// TwinCAT 3 PLC project plc_lamp_lv17_vac
// ProgramVersion: 3.1.4022.7
// CompilerDefines: VISU_USEPROPERTYINFO
// libraries:
//   LCLS General, * (SLAC)
//   PMPS, * (SLAC - LCLS)
//   Tc2_SerialCom, * (Beckhoff Automation GmbH)
//   Tc2_Standard, * (Beckhoff Automation GmbH)
//   Tc2_System, * (Beckhoff Automation GmbH)
//   Tc3_Module, * (Beckhoff Automation GmbH)
//   LCLS Vacuum,1.4.0,SLAC - LCLS
//   LCLSVacuumSerialDriverLib,1.2.2,SLAC - LCLS
// project tree:
//   / ComTask.TcTTO (not stored), GlobalTextList.TcGTLO (not stored), PlcTask.TcTTO (not stored)
//   GVLs/ GVL_COM.TcGVL, GVL_Devices.TcGVL, GVL_PLC_Interfaces.TcGVL (not stored), GVL_Variables.TcGVL (not stored)
//   POUs/ DIAGNOSTICS.TcPOU (not stored), F_Turbo_NC_NO_Valve_Logic.TcPOU (not stored), MAIN.TcPOU, PRG_COM.TcPOU
// real-time tasks:
//   TASK PlcTask: cycle T#10ms, priority 20, ADS port 350
//   TASK ComTask: cycle T#10ms, priority 15, ADS port 351
// I/O:
//   DEVICE Device 1 (EtherCAT), AmsNetId 172.21.132.34.2.1
//     LAMP_PLC_E0_EK1200 [EK1200-5000 EtherCAT Power supply (2A E-Bus)]
//       LAMP_PLC_E1_EL2202
//       LAMP_PLC_E2_EL6070
//       LAMP_PLC_E3_EL6692 [EL6692 EtherCAT Bridge terminal (Primary)]
//       LAMP_PLC_E4_EL9410
//       LAMP_PLC_E5_EL1004
//       LAMP_PLC_E6_EL2794
//       LAMP_PLC_E7_EL1004
//       LAMP_PLC_E8_EL2794
//       LAMP_PLC_E9_EL3318 [EL3318 8Ch. Ana Input Thermocouple (TC)]
//       LAMP_PLC_E10_EL6002
//       LAMP_PLC_E11_EL6002
//       LAMP_PLC_E12_EK1122 [EK1122 2 port EtherCAT junction]
//         LAMP_PNL_EP00_EP9128-0021 [EP9128-0021 8x EtherCAT junction]
//           LAMP_PNL1_EP01_EP2338-0002
//           LAMP_PNL1_EP02_EP2624-0002
//           LAMP_PNL1_EP03_EP6002-0002
//           LAMP_PNL1_EP04_EP2338-0002
//           LAMP_PNL1_EP05_EP2624-0002
//           LAMP_PNL1_EP06_EP6002-0002
//           LAMP_PNL1_EP07_EP2338-0002
//           LAMP_PNL1_EP08_EP2624-0002
//           LAMP_PNL1_EP09_EP6002-0002
//           LAMP_PNL1_EP10_EP2338-0002
//           LAMP_PNL1_EP11_EP2624-0002
//           LAMP_PNL1_EP12_EP6002-0002
//           LAMP_PNL2_EP13_EP2338-0002
//           LAMP_PNL2_EP14_EP2624-0002
//           LAMP_PNL2_EP15_EP6002-0002
//           LAMP_PNL2_EP16_EP2338-0002
//           LAMP_PNL2_EP17_EP2624-0002
//           LAMP_PN2_EP18_EP6002-0002
//           LAMP_PNL2_EP19_EP3174-0002
//           LAMP_PNL2_EP20_EP3174-0002
//           LAMP_PNL2_EP21_EP3174-0002
//           LAMP_PNL2_EP22_EP2624-0002
//           LAMP_PNL2_EP23_EP3174-0002
//           LAMP_PNL2_EP24_EP2624-0002
//           LAMP_PNL2_EP25_EP2338-0002
//           LAMP_PNL2_EP26_EP2338-0002
//           Term 88 (EP9128-1021) [EP9128-1021 8x EtherCAT junction - Dev A]
//             LAMP_CLSTR1_PNL1_EP01_EP2338-0002
//             LAMP_CLSTR1_PNL1_EP_02_EP2624-0002
//             LAMP_CLSTR1_PNL1_EP03_EP6002-0002
//             LAMP_CLSTR1_PNL3_EP01_EP2338-0002
//             LAMP_CLSTR1_PNL3_EP02_EP2624-0002
//             LAMP_CLSTR1_PNL3_EP03_EP6002-0002
//           Term 89 (EP9128-2021) [EP9128-2021 8x EtherCAT junction - Dev B]
//             LAMP_CLSTR1_PNL2_EP01_EP2338-0002
//             LAMP_CLSTR1_PNL2_EP02_EP2624-0002
//             LAMP_CLSTR1_PNL2_EP03_EP6002-0002
//             LAMP_CLSTR1_DCT_EP9224-0023
//         LAMP_PNL1_PWR_FOUT_Box (EP9224-0023) [EP9224-0023 4Ch/4Ch enhanced Power Distribution for EtherCAT Box Modules]
// variable links:
//   plc_lamp_lv17_vac/plc_lamp_lv17_vac Instance <-> Device 1 (EtherCAT)/LAMP_PLC_E0_EK1200/LAMP_PLC_E12_EK1122/LAMP_PNL_EP00_EP9128-0021/LAMP_PNL1_EP01_EP2338-0002
//     PlcTask Inputs/GVL_Devices.LAMP_C2_PTM_01.i_xAtSpd <-> Channel 1/Input
//     PlcTask Inputs/GVL_Devices.LAMP_C2_PTM_02.i_xAtSpd <-> Channel 5/Input
//     PlcTask Inputs/GVL_Devices.LAMP_C2_PTM_01.i_xFaultNC <-> Channel 2/Input
//     PlcTask Inputs/GVL_Devices.LAMP_C2_PTM_02.i_xFaultNC <-> Channel 6/Input
//     PlcTask Inputs/GVL_Devices.LAMP_C2_PTM_01.i_xRemote <-> Channel 3/Input
//     PlcTask Inputs/GVL_Devices.LAMP_C2_PTM_02.i_xRemote <-> Channel 7/Input
//   plc_lamp_lv17_vac/plc_lamp_lv17_vac Instance <-> Device 1 (EtherCAT)/LAMP_PLC_E0_EK1200/LAMP_PLC_E12_EK1122/LAMP_PNL_EP00_EP9128-0021/LAMP_PNL1_EP02_EP2624-0002
//     PlcTask Outputs/GVL_Devices.LAMP_C2_PTM_01.q_RunDO <-> Channel 1/Output
//     PlcTask Outputs/GVL_Devices.LAMP_C2_PTM_02.q_RunDO <-> Channel 3/Output
//     PlcTask Outputs/GVL_Devices.LAMP_C2_PTM_01.q_xReset <-> Channel 2/Output
//     PlcTask Outputs/GVL_Devices.LAMP_C2_PTM_02.q_xReset <-> Channel 4/Output
//   plc_lamp_lv17_vac/plc_lamp_lv17_vac Instance <-> Device 1 (EtherCAT)/LAMP_PLC_E0_EK1200/LAMP_PLC_E12_EK1122/LAMP_PNL_EP00_EP9128-0021/LAMP_PNL1_EP03_EP6002-0002
//     ComTask Inputs/GVL_COM.stComIn_LAMP_C2_PTM_01/D[0] <-> COM TxPDO-Map Inputs Channel 1/Data In 0
//     ComTask Inputs/GVL_COM.stComIn_LAMP_C2_PTM_01/D[10] <-> COM TxPDO-Map Inputs Channel 1/Data In 10
//     ComTask Inputs/GVL_COM.stComIn_LAMP_C2_PTM_01/D[11] <-> COM TxPDO-Map Inputs Channel 1/Data In 11
//     ComTask Inputs/GVL_COM.stComIn_LAMP_C2_PTM_01/D[12] <-> COM TxPDO-Map Inputs Channel 1/Data In 12
//     ComTask Inputs/GVL_COM.stComIn_LAMP_C2_PTM_01/D[13] <-> COM TxPDO-Map Inputs Channel 1/Data In 13
//     ComTask Inputs/GVL_COM.stComIn_LAMP_C2_PTM_01/D[14] <-> COM TxPDO-Map Inputs Channel 1/Data In 14
//     ComTask Inputs/GVL_COM.stComIn_LAMP_C2_PTM_01/D[15] <-> COM TxPDO-Map Inputs Channel 1/Data In 15
//     ComTask Inputs/GVL_COM.stComIn_LAMP_C2_PTM_01/D[16] <-> COM TxPDO-Map Inputs Channel 1/Data In 16
//     ComTask Inputs/GVL_COM.stComIn_LAMP_C2_PTM_01/D[17] <-> COM TxPDO-Map Inputs Channel 1/Data In 17
//     ComTask Inputs/GVL_COM.stComIn_LAMP_C2_PTM_01/D[18] <-> COM TxPDO-Map Inputs Channel 1/Data In 18
//     ComTask Inputs/GVL_COM.stComIn_LAMP_C2_PTM_01/D[19] <-> COM TxPDO-Map Inputs Channel 1/Data In 19
//     ComTask Inputs/GVL_COM.stComIn_LAMP_C2_PTM_01/D[1] <-> COM TxPDO-Map Inputs Channel 1/Data In 1
//     ComTask Inputs/GVL_COM.stComIn_LAMP_C2_PTM_01/D[20] <-> COM TxPDO-Map Inputs Channel 1/Data In 20
//     ComTask Inputs/GVL_COM.stComIn_LAMP_C2_PTM_01/D[21] <-> COM TxPDO-Map Inputs Channel 1/Data In 21
//     ComTask Inputs/GVL_COM.stComIn_LAMP_C2_PTM_01/D[2] <-> COM TxPDO-Map Inputs Channel 1/Data In 2
//     ComTask Inputs/GVL_COM.stComIn_LAMP_C2_PTM_01/D[3] <-> COM TxPDO-Map Inputs Channel 1/Data In 3
//     ComTask Inputs/GVL_COM.stComIn_LAMP_C2_PTM_01/D[4] <-> COM TxPDO-Map Inputs Channel 1/Data In 4
//     ComTask Inputs/GVL_COM.stComIn_LAMP_C2_PTM_01/D[5] <-> COM TxPDO-Map Inputs Channel 1/Data In 5
//     ComTask Inputs/GVL_COM.stComIn_LAMP_C2_PTM_01/D[6] <-> COM TxPDO-Map Inputs Channel 1/Data In 6
//     ComTask Inputs/GVL_COM.stComIn_LAMP_C2_PTM_01/D[7] <-> COM TxPDO-Map Inputs Channel 1/Data In 7
//     ComTask Inputs/GVL_COM.stComIn_LAMP_C2_PTM_01/D[8] <-> COM TxPDO-Map Inputs Channel 1/Data In 8
//     ComTask Inputs/GVL_COM.stComIn_LAMP_C2_PTM_01/D[9] <-> COM TxPDO-Map Inputs Channel 1/Data In 9
//     ComTask Inputs/GVL_COM.stComIn_LAMP_C2_PTM_02/D[0] <-> COM TxPDO-Map Inputs Channel 2/Data In 0
//     ComTask Inputs/GVL_COM.stComIn_LAMP_C2_PTM_02/D[10] <-> COM TxPDO-Map Inputs Channel 2/Data In 10
//     ComTask Inputs/GVL_COM.stComIn_LAMP_C2_PTM_02/D[11] <-> COM TxPDO-Map Inputs Channel 2/Data In 11
//     ComTask Inputs/GVL_COM.stComIn_LAMP_C2_PTM_02/D[12] <-> COM TxPDO-Map Inputs Channel 2/Data In 12
//     ComTask Inputs/GVL_COM.stComIn_LAMP_C2_PTM_02/D[13] <-> COM TxPDO-Map Inputs Channel 2/Data In 13
//     ComTask Inputs/GVL_COM.stComIn_LAMP_C2_PTM_02/D[14] <-> COM TxPDO-Map Inputs Channel 2/Data In 14
//     ComTask Inputs/GVL_COM.stComIn_LAMP_C2_PTM_02/D[15] <-> COM TxPDO-Map Inputs Channel 2/Data In 15
//     ComTask Inputs/GVL_COM.stComIn_LAMP_C2_PTM_02/D[16] <-> COM TxPDO-Map Inputs Channel 2/Data In 16
//     ComTask Inputs/GVL_COM.stComIn_LAMP_C2_PTM_02/D[17] <-> COM TxPDO-Map Inputs Channel 2/Data In 17
//     ComTask Inputs/GVL_COM.stComIn_LAMP_C2_PTM_02/D[18] <-> COM TxPDO-Map Inputs Channel 2/Data In 18
//     ComTask Inputs/GVL_COM.stComIn_LAMP_C2_PTM_02/D[19] <-> COM TxPDO-Map Inputs Channel 2/Data In 19
//     ComTask Inputs/GVL_COM.stComIn_LAMP_C2_PTM_02/D[1] <-> COM TxPDO-Map Inputs Channel 2/Data In 1
//     ComTask Inputs/GVL_COM.stComIn_LAMP_C2_PTM_02/D[20] <-> COM TxPDO-Map Inputs Channel 2/Data In 20
//     ComTask Inputs/GVL_COM.stComIn_LAMP_C2_PTM_02/D[21] <-> COM TxPDO-Map Inputs Channel 2/Data In 21
//     ComTask Inputs/GVL_COM.stComIn_LAMP_C2_PTM_02/D[2] <-> COM TxPDO-Map Inputs Channel 2/Data In 2
//     ComTask Inputs/GVL_COM.stComIn_LAMP_C2_PTM_02/D[3] <-> COM TxPDO-Map Inputs Channel 2/Data In 3
//     ComTask Inputs/GVL_COM.stComIn_LAMP_C2_PTM_02/D[4] <-> COM TxPDO-Map Inputs Channel 2/Data In 4
//     ComTask Inputs/GVL_COM.stComIn_LAMP_C2_PTM_02/D[5] <-> COM TxPDO-Map Inputs Channel 2/Data In 5
//     ComTask Inputs/GVL_COM.stComIn_LAMP_C2_PTM_02/D[6] <-> COM TxPDO-Map Inputs Channel 2/Data In 6
//     ComTask Inputs/GVL_COM.stComIn_LAMP_C2_PTM_02/D[7] <-> COM TxPDO-Map Inputs Channel 2/Data In 7
//     ComTask Inputs/GVL_COM.stComIn_LAMP_C2_PTM_02/D[8] <-> COM TxPDO-Map Inputs Channel 2/Data In 8
//     ComTask Inputs/GVL_COM.stComIn_LAMP_C2_PTM_02/D[9] <-> COM TxPDO-Map Inputs Channel 2/Data In 9
//     ComTask Inputs/GVL_COM.stComIn_LAMP_C2_PTM_01/Status <-> COM TxPDO-Map Inputs Channel 1/Status
//     ComTask Inputs/GVL_COM.stComIn_LAMP_C2_PTM_02/Status <-> COM TxPDO-Map Inputs Channel 2/Status
//     ComTask Outputs/GVL_COM.stComOut_LAMP_C2_PTM_01/Ctrl <-> COM RxPDO-Map Outputs Channel 1/Ctrl
//     ComTask Outputs/GVL_COM.stComOut_LAMP_C2_PTM_02/Ctrl <-> COM RxPDO-Map Outputs Channel 2/Ctrl
//     ComTask Outputs/GVL_COM.stComOut_LAMP_C2_PTM_01/D[0] <-> COM RxPDO-Map Outputs Channel 1/Data Out 0
//     ComTask Outputs/GVL_COM.stComOut_LAMP_C2_PTM_01/D[10] <-> COM RxPDO-Map Outputs Channel 1/Data Out 10
//     ComTask Outputs/GVL_COM.stComOut_LAMP_C2_PTM_01/D[11] <-> COM RxPDO-Map Outputs Channel 1/Data Out 11
//     ComTask Outputs/GVL_COM.stComOut_LAMP_C2_PTM_01/D[12] <-> COM RxPDO-Map Outputs Channel 1/Data Out 12
//     ComTask Outputs/GVL_COM.stComOut_LAMP_C2_PTM_01/D[13] <-> COM RxPDO-Map Outputs Channel 1/Data Out 13
//     ComTask Outputs/GVL_COM.stComOut_LAMP_C2_PTM_01/D[14] <-> COM RxPDO-Map Outputs Channel 1/Data Out 14
//     ComTask Outputs/GVL_COM.stComOut_LAMP_C2_PTM_01/D[15] <-> COM RxPDO-Map Outputs Channel 1/Data Out 15
//     ComTask Outputs/GVL_COM.stComOut_LAMP_C2_PTM_01/D[16] <-> COM RxPDO-Map Outputs Channel 1/Data Out 16
//     ComTask Outputs/GVL_COM.stComOut_LAMP_C2_PTM_01/D[17] <-> COM RxPDO-Map Outputs Channel 1/Data Out 17
//     ComTask Outputs/GVL_COM.stComOut_LAMP_C2_PTM_01/D[18] <-> COM RxPDO-Map Outputs Channel 1/Data Out 18
//     ComTask Outputs/GVL_COM.stComOut_LAMP_C2_PTM_01/D[19] <-> COM RxPDO-Map Outputs Channel 1/Data Out 19
//     ComTask Outputs/GVL_COM.stComOut_LAMP_C2_PTM_01/D[1] <-> COM RxPDO-Map Outputs Channel 1/Data Out 1
//     ComTask Outputs/GVL_COM.stComOut_LAMP_C2_PTM_01/D[20] <-> COM RxPDO-Map Outputs Channel 1/Data Out 20
//     ComTask Outputs/GVL_COM.stComOut_LAMP_C2_PTM_01/D[21] <-> COM RxPDO-Map Outputs Channel 1/Data Out 21
//     ComTask Outputs/GVL_COM.stComOut_LAMP_C2_PTM_01/D[2] <-> COM RxPDO-Map Outputs Channel 1/Data Out 2
//     ComTask Outputs/GVL_COM.stComOut_LAMP_C2_PTM_01/D[3] <-> COM RxPDO-Map Outputs Channel 1/Data Out 3
//     ComTask Outputs/GVL_COM.stComOut_LAMP_C2_PTM_01/D[4] <-> COM RxPDO-Map Outputs Channel 1/Data Out 4
//     ComTask Outputs/GVL_COM.stComOut_LAMP_C2_PTM_01/D[5] <-> COM RxPDO-Map Outputs Channel 1/Data Out 5
//     ComTask Outputs/GVL_COM.stComOut_LAMP_C2_PTM_01/D[6] <-> COM RxPDO-Map Outputs Channel 1/Data Out 6
//     ComTask Outputs/GVL_COM.stComOut_LAMP_C2_PTM_01/D[7] <-> COM RxPDO-Map Outputs Channel 1/Data Out 7
//     ComTask Outputs/GVL_COM.stComOut_LAMP_C2_PTM_01/D[8] <-> COM RxPDO-Map Outputs Channel 1/Data Out 8
//     ComTask Outputs/GVL_COM.stComOut_LAMP_C2_PTM_01/D[9] <-> COM RxPDO-Map Outputs Channel 1/Data Out 9
//     ComTask Outputs/GVL_COM.stComOut_LAMP_C2_PTM_02/D[0] <-> COM RxPDO-Map Outputs Channel 2/Data Out 0
//     ComTask Outputs/GVL_COM.stComOut_LAMP_C2_PTM_02/D[10] <-> COM RxPDO-Map Outputs Channel 2/Data Out 10
//     ComTask Outputs/GVL_COM.stComOut_LAMP_C2_PTM_02/D[11] <-> COM RxPDO-Map Outputs Channel 2/Data Out 11
//     ComTask Outputs/GVL_COM.stComOut_LAMP_C2_PTM_02/D[12] <-> COM RxPDO-Map Outputs Channel 2/Data Out 12
//     ComTask Outputs/GVL_COM.stComOut_LAMP_C2_PTM_02/D[13] <-> COM RxPDO-Map Outputs Channel 2/Data Out 13
//     ComTask Outputs/GVL_COM.stComOut_LAMP_C2_PTM_02/D[14] <-> COM RxPDO-Map Outputs Channel 2/Data Out 14
//     ComTask Outputs/GVL_COM.stComOut_LAMP_C2_PTM_02/D[15] <-> COM RxPDO-Map Outputs Channel 2/Data Out 15
//     ComTask Outputs/GVL_COM.stComOut_LAMP_C2_PTM_02/D[16] <-> COM RxPDO-Map Outputs Channel 2/Data Out 16
//     ComTask Outputs/GVL_COM.stComOut_LAMP_C2_PTM_02/D[17] <-> COM RxPDO-Map Outputs Channel 2/Data Out 17
//     ComTask Outputs/GVL_COM.stComOut_LAMP_C2_PTM_02/D[18] <-> COM RxPDO-Map Outputs Channel 2/Data Out 18
//     ComTask Outputs/GVL_COM.stComOut_LAMP_C2_PTM_02/D[19] <-> COM RxPDO-Map Outputs Channel 2/Data Out 19
//     ComTask Outputs/GVL_COM.stComOut_LAMP_C2_PTM_02/D[1] <-> COM RxPDO-Map Outputs Channel 2/Data Out 1
//     ComTask Outputs/GVL_COM.stComOut_LAMP_C2_PTM_02/D[20] <-> COM RxPDO-Map Outputs Channel 2/Data Out 20
//     ComTask Outputs/GVL_COM.stComOut_LAMP_C2_PTM_02/D[21] <-> COM RxPDO-Map Outputs Channel 2/Data Out 21
//     ComTask Outputs/GVL_COM.stComOut_LAMP_C2_PTM_02/D[2] <-> COM RxPDO-Map Outputs Channel 2/Data Out 2
//     ComTask Outputs/GVL_COM.stComOut_LAMP_C2_PTM_02/D[3] <-> COM RxPDO-Map Outputs Channel 2/Data Out 3
//     ComTask Outputs/GVL_COM.stComOut_LAMP_C2_PTM_02/D[4] <-> COM RxPDO-Map Outputs Channel 2/Data Out 4
//     ComTask Outputs/GVL_COM.stComOut_LAMP_C2_PTM_02/D[5] <-> COM RxPDO-Map Outputs Channel 2/Data Out 5
//     ComTask Outputs/GVL_COM.stComOut_LAMP_C2_PTM_02/D[6] <-> COM RxPDO-Map Outputs Channel 2/Data Out 6
//     ComTask Outputs/GVL_COM.stComOut_LAMP_C2_PTM_02/D[7] <-> COM RxPDO-Map Outputs Channel 2/Data Out 7
//     ComTask Outputs/GVL_COM.stComOut_LAMP_C2_PTM_02/D[8] <-> COM RxPDO-Map Outputs Channel 2/Data Out 8
//     ComTask Outputs/GVL_COM.stComOut_LAMP_C2_PTM_02/D[9] <-> COM RxPDO-Map Outputs Channel 2/Data Out 9
//   plc_lamp_lv17_vac/plc_lamp_lv17_vac Instance <-> Device 1 (EtherCAT)/LAMP_PLC_E0_EK1200/LAMP_PLC_E12_EK1122/LAMP_PNL_EP00_EP9128-0021/LAMP_PNL1_EP04_EP2338-0002
//     PlcTask Inputs/GVL_Devices.LAMP_C2_PTM_03.i_xAtSpd <-> Channel 1/Input
//     PlcTask Inputs/GVL_Devices.LAMP_C2_PTM_04.i_xAtSpd <-> Channel 5/Input
//     PlcTask Inputs/GVL_Devices.LAMP_C2_PTM_03.i_xFaultNC <-> Channel 2/Input
//     PlcTask Inputs/GVL_Devices.LAMP_C2_PTM_04.i_xFaultNC <-> Channel 6/Input
//     PlcTask Inputs/GVL_Devices.LAMP_C2_PTM_03.i_xRemote <-> Channel 3/Input
//     PlcTask Inputs/GVL_Devices.LAMP_C2_PTM_04.i_xRemote <-> Channel 7/Input
//   plc_lamp_lv17_vac/plc_lamp_lv17_vac Instance <-> Device 1 (EtherCAT)/LAMP_PLC_E0_EK1200/LAMP_PLC_E12_EK1122/LAMP_PNL_EP00_EP9128-0021/LAMP_PNL1_EP05_EP2624-0002
//     PlcTask Outputs/GVL_Devices.LAMP_C2_PTM_03.q_RunDO <-> Channel 1/Output
//     PlcTask Outputs/GVL_Devices.LAMP_C2_PTM_04.q_RunDO <-> Channel 3/Output
//     PlcTask Outputs/GVL_Devices.LAMP_C2_PTM_03.q_xReset <-> Channel 2/Output
//     PlcTask Outputs/GVL_Devices.LAMP_C2_PTM_04.q_xReset <-> Channel 4/Output
//   plc_lamp_lv17_vac/plc_lamp_lv17_vac Instance <-> Device 1 (EtherCAT)/LAMP_PLC_E0_EK1200/LAMP_PLC_E12_EK1122/LAMP_PNL_EP00_EP9128-0021/LAMP_PNL1_EP06_EP6002-0002
//     ComTask Inputs/GVL_COM.stComIn_LAMP_C2_PTM_03/D[0] <-> COM TxPDO-Map Inputs Channel 1/Data In 0
//     ComTask Inputs/GVL_COM.stComIn_LAMP_C2_PTM_03/D[10] <-> COM TxPDO-Map Inputs Channel 1/Data In 10
//     ComTask Inputs/GVL_COM.stComIn_LAMP_C2_PTM_03/D[11] <-> COM TxPDO-Map Inputs Channel 1/Data In 11
//     ComTask Inputs/GVL_COM.stComIn_LAMP_C2_PTM_03/D[12] <-> COM TxPDO-Map Inputs Channel 1/Data In 12
//     ComTask Inputs/GVL_COM.stComIn_LAMP_C2_PTM_03/D[13] <-> COM TxPDO-Map Inputs Channel 1/Data In 13
//     ComTask Inputs/GVL_COM.stComIn_LAMP_C2_PTM_03/D[14] <-> COM TxPDO-Map Inputs Channel 1/Data In 14
//     ComTask Inputs/GVL_COM.stComIn_LAMP_C2_PTM_03/D[15] <-> COM TxPDO-Map Inputs Channel 1/Data In 15
//     ComTask Inputs/GVL_COM.stComIn_LAMP_C2_PTM_03/D[16] <-> COM TxPDO-Map Inputs Channel 1/Data In 16
//     ComTask Inputs/GVL_COM.stComIn_LAMP_C2_PTM_03/D[17] <-> COM TxPDO-Map Inputs Channel 1/Data In 17
//     ComTask Inputs/GVL_COM.stComIn_LAMP_C2_PTM_03/D[18] <-> COM TxPDO-Map Inputs Channel 1/Data In 18
//     ComTask Inputs/GVL_COM.stComIn_LAMP_C2_PTM_03/D[19] <-> COM TxPDO-Map Inputs Channel 1/Data In 19
//     ComTask Inputs/GVL_COM.stComIn_LAMP_C2_PTM_03/D[1] <-> COM TxPDO-Map Inputs Channel 1/Data In 1
//     ComTask Inputs/GVL_COM.stComIn_LAMP_C2_PTM_03/D[20] <-> COM TxPDO-Map Inputs Channel 1/Data In 20
//     ComTask Inputs/GVL_COM.stComIn_LAMP_C2_PTM_03/D[21] <-> COM TxPDO-Map Inputs Channel 1/Data In 21
//     ComTask Inputs/GVL_COM.stComIn_LAMP_C2_PTM_03/D[2] <-> COM TxPDO-Map Inputs Channel 1/Data In 2
//     ComTask Inputs/GVL_COM.stComIn_LAMP_C2_PTM_03/D[3] <-> COM TxPDO-Map Inputs Channel 1/Data In 3
//     ComTask Inputs/GVL_COM.stComIn_LAMP_C2_PTM_03/D[4] <-> COM TxPDO-Map Inputs Channel 1/Data In 4
//     ComTask Inputs/GVL_COM.stComIn_LAMP_C2_PTM_03/D[5] <-> COM TxPDO-Map Inputs Channel 1/Data In 5
//     ComTask Inputs/GVL_COM.stComIn_LAMP_C2_PTM_03/D[6] <-> COM TxPDO-Map Inputs Channel 1/Data In 6
//     ComTask Inputs/GVL_COM.stComIn_LAMP_C2_PTM_03/D[7] <-> COM TxPDO-Map Inputs Channel 1/Data In 7
//     ComTask Inputs/GVL_COM.stComIn_LAMP_C2_PTM_03/D[8] <-> COM TxPDO-Map Inputs Channel 1/Data In 8
//     ComTask Inputs/GVL_COM.stComIn_LAMP_C2_PTM_03/D[9] <-> COM TxPDO-Map Inputs Channel 1/Data In 9
//     ComTask Inputs/GVL_COM.stComIn_LAMP_C2_PTM_04/D[0] <-> COM TxPDO-Map Inputs Channel 2/Data In 0
//     ComTask Inputs/GVL_COM.stComIn_LAMP_C2_PTM_04/D[10] <-> COM TxPDO-Map Inputs Channel 2/Data In 10
//     ComTask Inputs/GVL_COM.stComIn_LAMP_C2_PTM_04/D[11] <-> COM TxPDO-Map Inputs Channel 2/Data In 11
//     ComTask Inputs/GVL_COM.stComIn_LAMP_C2_PTM_04/D[12] <-> COM TxPDO-Map Inputs Channel 2/Data In 12
//     ComTask Inputs/GVL_COM.stComIn_LAMP_C2_PTM_04/D[13] <-> COM TxPDO-Map Inputs Channel 2/Data In 13
//     ComTask Inputs/GVL_COM.stComIn_LAMP_C2_PTM_04/D[14] <-> COM TxPDO-Map Inputs Channel 2/Data In 14
//     ComTask Inputs/GVL_COM.stComIn_LAMP_C2_PTM_04/D[15] <-> COM TxPDO-Map Inputs Channel 2/Data In 15
//     ComTask Inputs/GVL_COM.stComIn_LAMP_C2_PTM_04/D[16] <-> COM TxPDO-Map Inputs Channel 2/Data In 16
//     ComTask Inputs/GVL_COM.stComIn_LAMP_C2_PTM_04/D[17] <-> COM TxPDO-Map Inputs Channel 2/Data In 17
//     ComTask Inputs/GVL_COM.stComIn_LAMP_C2_PTM_04/D[18] <-> COM TxPDO-Map Inputs Channel 2/Data In 18
//     ComTask Inputs/GVL_COM.stComIn_LAMP_C2_PTM_04/D[19] <-> COM TxPDO-Map Inputs Channel 2/Data In 19
//     ComTask Inputs/GVL_COM.stComIn_LAMP_C2_PTM_04/D[1] <-> COM TxPDO-Map Inputs Channel 2/Data In 1
//     ComTask Inputs/GVL_COM.stComIn_LAMP_C2_PTM_04/D[20] <-> COM TxPDO-Map Inputs Channel 2/Data In 20
//     ComTask Inputs/GVL_COM.stComIn_LAMP_C2_PTM_04/D[21] <-> COM TxPDO-Map Inputs Channel 2/Data In 21
//     ComTask Inputs/GVL_COM.stComIn_LAMP_C2_PTM_04/D[2] <-> COM TxPDO-Map Inputs Channel 2/Data In 2
//     ComTask Inputs/GVL_COM.stComIn_LAMP_C2_PTM_04/D[3] <-> COM TxPDO-Map Inputs Channel 2/Data In 3
//     ComTask Inputs/GVL_COM.stComIn_LAMP_C2_PTM_04/D[4] <-> COM TxPDO-Map Inputs Channel 2/Data In 4
//     ComTask Inputs/GVL_COM.stComIn_LAMP_C2_PTM_04/D[5] <-> COM TxPDO-Map Inputs Channel 2/Data In 5
//     ComTask Inputs/GVL_COM.stComIn_LAMP_C2_PTM_04/D[6] <-> COM TxPDO-Map Inputs Channel 2/Data In 6
//     ComTask Inputs/GVL_COM.stComIn_LAMP_C2_PTM_04/D[7] <-> COM TxPDO-Map Inputs Channel 2/Data In 7
//     ComTask Inputs/GVL_COM.stComIn_LAMP_C2_PTM_04/D[8] <-> COM TxPDO-Map Inputs Channel 2/Data In 8
//     ComTask Inputs/GVL_COM.stComIn_LAMP_C2_PTM_04/D[9] <-> COM TxPDO-Map Inputs Channel 2/Data In 9
//     ComTask Inputs/GVL_COM.stComIn_LAMP_C2_PTM_03/Status <-> COM TxPDO-Map Inputs Channel 1/Status
//     ComTask Inputs/GVL_COM.stComIn_LAMP_C2_PTM_04/Status <-> COM TxPDO-Map Inputs Channel 2/Status
//     ComTask Outputs/GVL_COM.stComOut_LAMP_C2_PTM_03/Ctrl <-> COM RxPDO-Map Outputs Channel 1/Ctrl
//     ComTask Outputs/GVL_COM.stComOut_LAMP_C2_PTM_04/Ctrl <-> COM RxPDO-Map Outputs Channel 2/Ctrl
//     ComTask Outputs/GVL_COM.stComOut_LAMP_C2_PTM_03/D[0] <-> COM RxPDO-Map Outputs Channel 1/Data Out 0
//     ComTask Outputs/GVL_COM.stComOut_LAMP_C2_PTM_03/D[10] <-> COM RxPDO-Map Outputs Channel 1/Data Out 10
//     ComTask Outputs/GVL_COM.stComOut_LAMP_C2_PTM_03/D[11] <-> COM RxPDO-Map Outputs Channel 1/Data Out 11
//     ComTask Outputs/GVL_COM.stComOut_LAMP_C2_PTM_03/D[12] <-> COM RxPDO-Map Outputs Channel 1/Data Out 12
//     ComTask Outputs/GVL_COM.stComOut_LAMP_C2_PTM_03/D[13] <-> COM RxPDO-Map Outputs Channel 1/Data Out 13
//     ComTask Outputs/GVL_COM.stComOut_LAMP_C2_PTM_03/D[14] <-> COM RxPDO-Map Outputs Channel 1/Data Out 14
//     ComTask Outputs/GVL_COM.stComOut_LAMP_C2_PTM_03/D[15] <-> COM RxPDO-Map Outputs Channel 1/Data Out 15
//     ComTask Outputs/GVL_COM.stComOut_LAMP_C2_PTM_03/D[16] <-> COM RxPDO-Map Outputs Channel 1/Data Out 16
//     ComTask Outputs/GVL_COM.stComOut_LAMP_C2_PTM_03/D[17] <-> COM RxPDO-Map Outputs Channel 1/Data Out 17
//     ComTask Outputs/GVL_COM.stComOut_LAMP_C2_PTM_03/D[18] <-> COM RxPDO-Map Outputs Channel 1/Data Out 18
//     ComTask Outputs/GVL_COM.stComOut_LAMP_C2_PTM_03/D[19] <-> COM RxPDO-Map Outputs Channel 1/Data Out 19
//     ComTask Outputs/GVL_COM.stComOut_LAMP_C2_PTM_03/D[1] <-> COM RxPDO-Map Outputs Channel 1/Data Out 1
//     ComTask Outputs/GVL_COM.stComOut_LAMP_C2_PTM_03/D[20] <-> COM RxPDO-Map Outputs Channel 1/Data Out 20
//     ComTask Outputs/GVL_COM.stComOut_LAMP_C2_PTM_03/D[21] <-> COM RxPDO-Map Outputs Channel 1/Data Out 21
//     ComTask Outputs/GVL_COM.stComOut_LAMP_C2_PTM_03/D[2] <-> COM RxPDO-Map Outputs Channel 1/Data Out 2
//     ComTask Outputs/GVL_COM.stComOut_LAMP_C2_PTM_03/D[3] <-> COM RxPDO-Map Outputs Channel 1/Data Out 3
//     ComTask Outputs/GVL_COM.stComOut_LAMP_C2_PTM_03/D[4] <-> COM RxPDO-Map Outputs Channel 1/Data Out 4
//     ComTask Outputs/GVL_COM.stComOut_LAMP_C2_PTM_03/D[5] <-> COM RxPDO-Map Outputs Channel 1/Data Out 5
//     ComTask Outputs/GVL_COM.stComOut_LAMP_C2_PTM_03/D[6] <-> COM RxPDO-Map Outputs Channel 1/Data Out 6
//     ComTask Outputs/GVL_COM.stComOut_LAMP_C2_PTM_03/D[7] <-> COM RxPDO-Map Outputs Channel 1/Data Out 7
//     ComTask Outputs/GVL_COM.stComOut_LAMP_C2_PTM_03/D[8] <-> COM RxPDO-Map Outputs Channel 1/Data Out 8
//     ComTask Outputs/GVL_COM.stComOut_LAMP_C2_PTM_03/D[9] <-> COM RxPDO-Map Outputs Channel 1/Data Out 9
//     ComTask Outputs/GVL_COM.stComOut_LAMP_C2_PTM_04/D[0] <-> COM RxPDO-Map Outputs Channel 2/Data Out 0
//     ComTask Outputs/GVL_COM.stComOut_LAMP_C2_PTM_04/D[10] <-> COM RxPDO-Map Outputs Channel 2/Data Out 10
//     ComTask Outputs/GVL_COM.stComOut_LAMP_C2_PTM_04/D[11] <-> COM RxPDO-Map Outputs Channel 2/Data Out 11
//     ComTask Outputs/GVL_COM.stComOut_LAMP_C2_PTM_04/D[12] <-> COM RxPDO-Map Outputs Channel 2/Data Out 12
//     ComTask Outputs/GVL_COM.stComOut_LAMP_C2_PTM_04/D[13] <-> COM RxPDO-Map Outputs Channel 2/Data Out 13
//     ComTask Outputs/GVL_COM.stComOut_LAMP_C2_PTM_04/D[14] <-> COM RxPDO-Map Outputs Channel 2/Data Out 14
//     ComTask Outputs/GVL_COM.stComOut_LAMP_C2_PTM_04/D[15] <-> COM RxPDO-Map Outputs Channel 2/Data Out 15
//     ComTask Outputs/GVL_COM.stComOut_LAMP_C2_PTM_04/D[16] <-> COM RxPDO-Map Outputs Channel 2/Data Out 16
//     ComTask Outputs/GVL_COM.stComOut_LAMP_C2_PTM_04/D[17] <-> COM RxPDO-Map Outputs Channel 2/Data Out 17
//     ComTask Outputs/GVL_COM.stComOut_LAMP_C2_PTM_04/D[18] <-> COM RxPDO-Map Outputs Channel 2/Data Out 18
//     ComTask Outputs/GVL_COM.stComOut_LAMP_C2_PTM_04/D[19] <-> COM RxPDO-Map Outputs Channel 2/Data Out 19
//     ComTask Outputs/GVL_COM.stComOut_LAMP_C2_PTM_04/D[1] <-> COM RxPDO-Map Outputs Channel 2/Data Out 1
//     ComTask Outputs/GVL_COM.stComOut_LAMP_C2_PTM_04/D[20] <-> COM RxPDO-Map Outputs Channel 2/Data Out 20
//     ComTask Outputs/GVL_COM.stComOut_LAMP_C2_PTM_04/D[21] <-> COM RxPDO-Map Outputs Channel 2/Data Out 21
//     ComTask Outputs/GVL_COM.stComOut_LAMP_C2_PTM_04/D[2] <-> COM RxPDO-Map Outputs Channel 2/Data Out 2
//     ComTask Outputs/GVL_COM.stComOut_LAMP_C2_PTM_04/D[3] <-> COM RxPDO-Map Outputs Channel 2/Data Out 3
//     ComTask Outputs/GVL_COM.stComOut_LAMP_C2_PTM_04/D[4] <-> COM RxPDO-Map Outputs Channel 2/Data Out 4
//     ComTask Outputs/GVL_COM.stComOut_LAMP_C2_PTM_04/D[5] <-> COM RxPDO-Map Outputs Channel 2/Data Out 5
//     ComTask Outputs/GVL_COM.stComOut_LAMP_C2_PTM_04/D[6] <-> COM RxPDO-Map Outputs Channel 2/Data Out 6
//     ComTask Outputs/GVL_COM.stComOut_LAMP_C2_PTM_04/D[7] <-> COM RxPDO-Map Outputs Channel 2/Data Out 7
//     ComTask Outputs/GVL_COM.stComOut_LAMP_C2_PTM_04/D[8] <-> COM RxPDO-Map Outputs Channel 2/Data Out 8
//     ComTask Outputs/GVL_COM.stComOut_LAMP_C2_PTM_04/D[9] <-> COM RxPDO-Map Outputs Channel 2/Data Out 9
//   plc_lamp_lv17_vac/plc_lamp_lv17_vac Instance <-> Device 1 (EtherCAT)/LAMP_PLC_E0_EK1200/LAMP_PLC_E12_EK1122/LAMP_PNL_EP00_EP9128-0021/LAMP_PNL2_EP13_EP2338-0002
//     PlcTask Inputs/GVL_Devices.LAMP_C1_PTM_01.i_xAtSpd <-> Channel 5/Input
//     PlcTask Inputs/GVL_Devices.LAMP_C1_PTM_01.i_xFaultNC <-> Channel 6/Input
//     PlcTask Inputs/GVL_Devices.LAMP_C1_PTM_01.i_xRemote <-> Channel 7/Input
//     PlcTask Inputs/GVL_Devices.LAMP_ROUGH_PTM_01.i_xAtSpd <-> Channel 1/Input
//     PlcTask Inputs/GVL_Devices.LAMP_ROUGH_PTM_01.i_xFaultNC <-> Channel 2/Input
//     PlcTask Inputs/GVL_Devices.LAMP_ROUGH_PTM_01.i_xRemote <-> Channel 3/Input
//   plc_lamp_lv17_vac/plc_lamp_lv17_vac Instance <-> Device 1 (EtherCAT)/LAMP_PLC_E0_EK1200/LAMP_PLC_E12_EK1122/LAMP_PNL_EP00_EP9128-0021/LAMP_PNL2_EP14_EP2624-0002
//     PlcTask Outputs/GVL_Devices.LAMP_C1_PTM_01.q_RunDO <-> Channel 3/Output
//     PlcTask Outputs/GVL_Devices.LAMP_C1_PTM_01.q_xReset <-> Channel 4/Output
//     PlcTask Outputs/GVL_Devices.LAMP_ROUGH_PTM_01.q_RunDO <-> Channel 1/Output
//     PlcTask Outputs/GVL_Devices.LAMP_ROUGH_PTM_01.q_xReset <-> Channel 2/Output
//   plc_lamp_lv17_vac/plc_lamp_lv17_vac Instance <-> Device 1 (EtherCAT)/LAMP_PLC_E0_EK1200/LAMP_PLC_E12_EK1122/LAMP_PNL_EP00_EP9128-0021/LAMP_PNL2_EP15_EP6002-0002
//     ComTask Inputs/GVL_COM.stComIn_LAMP_C1_PTM_01/D[0] <-> COM TxPDO-Map Inputs Channel 2/Data In 0
//     ComTask Inputs/GVL_COM.stComIn_LAMP_C1_PTM_01/D[10] <-> COM TxPDO-Map Inputs Channel 2/Data In 10
//     ComTask Inputs/GVL_COM.stComIn_LAMP_C1_PTM_01/D[11] <-> COM TxPDO-Map Inputs Channel 2/Data In 11
//     ComTask Inputs/GVL_COM.stComIn_LAMP_C1_PTM_01/D[12] <-> COM TxPDO-Map Inputs Channel 2/Data In 12
//     ComTask Inputs/GVL_COM.stComIn_LAMP_C1_PTM_01/D[13] <-> COM TxPDO-Map Inputs Channel 2/Data In 13
//     ComTask Inputs/GVL_COM.stComIn_LAMP_C1_PTM_01/D[14] <-> COM TxPDO-Map Inputs Channel 2/Data In 14
//     ComTask Inputs/GVL_COM.stComIn_LAMP_C1_PTM_01/D[15] <-> COM TxPDO-Map Inputs Channel 2/Data In 15
//     ComTask Inputs/GVL_COM.stComIn_LAMP_C1_PTM_01/D[16] <-> COM TxPDO-Map Inputs Channel 2/Data In 16
//     ComTask Inputs/GVL_COM.stComIn_LAMP_C1_PTM_01/D[17] <-> COM TxPDO-Map Inputs Channel 2/Data In 17
//     ComTask Inputs/GVL_COM.stComIn_LAMP_C1_PTM_01/D[18] <-> COM TxPDO-Map Inputs Channel 2/Data In 18
//     ComTask Inputs/GVL_COM.stComIn_LAMP_C1_PTM_01/D[19] <-> COM TxPDO-Map Inputs Channel 2/Data In 19
//     ComTask Inputs/GVL_COM.stComIn_LAMP_C1_PTM_01/D[1] <-> COM TxPDO-Map Inputs Channel 2/Data In 1
//     ComTask Inputs/GVL_COM.stComIn_LAMP_C1_PTM_01/D[20] <-> COM TxPDO-Map Inputs Channel 2/Data In 20
//     ComTask Inputs/GVL_COM.stComIn_LAMP_C1_PTM_01/D[21] <-> COM TxPDO-Map Inputs Channel 2/Data In 21
//     ComTask Inputs/GVL_COM.stComIn_LAMP_C1_PTM_01/D[2] <-> COM TxPDO-Map Inputs Channel 2/Data In 2
//     ComTask Inputs/GVL_COM.stComIn_LAMP_C1_PTM_01/D[3] <-> COM TxPDO-Map Inputs Channel 2/Data In 3
//     ComTask Inputs/GVL_COM.stComIn_LAMP_C1_PTM_01/D[4] <-> COM TxPDO-Map Inputs Channel 2/Data In 4
//     ComTask Inputs/GVL_COM.stComIn_LAMP_C1_PTM_01/D[5] <-> COM TxPDO-Map Inputs Channel 2/Data In 5
//     ComTask Inputs/GVL_COM.stComIn_LAMP_C1_PTM_01/D[6] <-> COM TxPDO-Map Inputs Channel 2/Data In 6
//     ComTask Inputs/GVL_COM.stComIn_LAMP_C1_PTM_01/D[7] <-> COM TxPDO-Map Inputs Channel 2/Data In 7
//     ComTask Inputs/GVL_COM.stComIn_LAMP_C1_PTM_01/D[8] <-> COM TxPDO-Map Inputs Channel 2/Data In 8
//     ComTask Inputs/GVL_COM.stComIn_LAMP_C1_PTM_01/D[9] <-> COM TxPDO-Map Inputs Channel 2/Data In 9
//     ComTask Inputs/GVL_COM.stComIn_LAMP_C1_PTM_01/Status <-> COM TxPDO-Map Inputs Channel 2/Status
//     ComTask Inputs/GVL_COM.stComIn_LAMP_ROUGH_PTM_01/D[0] <-> COM TxPDO-Map Inputs Channel 1/Data In 0
//     ComTask Inputs/GVL_COM.stComIn_LAMP_ROUGH_PTM_01/D[10] <-> COM TxPDO-Map Inputs Channel 1/Data In 10
//     ComTask Inputs/GVL_COM.stComIn_LAMP_ROUGH_PTM_01/D[11] <-> COM TxPDO-Map Inputs Channel 1/Data In 11
//     ComTask Inputs/GVL_COM.stComIn_LAMP_ROUGH_PTM_01/D[12] <-> COM TxPDO-Map Inputs Channel 1/Data In 12
//     ComTask Inputs/GVL_COM.stComIn_LAMP_ROUGH_PTM_01/D[13] <-> COM TxPDO-Map Inputs Channel 1/Data In 13
//     ComTask Inputs/GVL_COM.stComIn_LAMP_ROUGH_PTM_01/D[14] <-> COM TxPDO-Map Inputs Channel 1/Data In 14
//     ComTask Inputs/GVL_COM.stComIn_LAMP_ROUGH_PTM_01/D[15] <-> COM TxPDO-Map Inputs Channel 1/Data In 15
//     ComTask Inputs/GVL_COM.stComIn_LAMP_ROUGH_PTM_01/D[16] <-> COM TxPDO-Map Inputs Channel 1/Data In 16
//     ComTask Inputs/GVL_COM.stComIn_LAMP_ROUGH_PTM_01/D[17] <-> COM TxPDO-Map Inputs Channel 1/Data In 17
//     ComTask Inputs/GVL_COM.stComIn_LAMP_ROUGH_PTM_01/D[18] <-> COM TxPDO-Map Inputs Channel 1/Data In 18
//     ComTask Inputs/GVL_COM.stComIn_LAMP_ROUGH_PTM_01/D[19] <-> COM TxPDO-Map Inputs Channel 1/Data In 19
//     ComTask Inputs/GVL_COM.stComIn_LAMP_ROUGH_PTM_01/D[1] <-> COM TxPDO-Map Inputs Channel 1/Data In 1
//     ComTask Inputs/GVL_COM.stComIn_LAMP_ROUGH_PTM_01/D[20] <-> COM TxPDO-Map Inputs Channel 1/Data In 20
//     ComTask Inputs/GVL_COM.stComIn_LAMP_ROUGH_PTM_01/D[21] <-> COM TxPDO-Map Inputs Channel 1/Data In 21
//     ComTask Inputs/GVL_COM.stComIn_LAMP_ROUGH_PTM_01/D[2] <-> COM TxPDO-Map Inputs Channel 1/Data In 2
//     ComTask Inputs/GVL_COM.stComIn_LAMP_ROUGH_PTM_01/D[3] <-> COM TxPDO-Map Inputs Channel 1/Data In 3
//     ComTask Inputs/GVL_COM.stComIn_LAMP_ROUGH_PTM_01/D[4] <-> COM TxPDO-Map Inputs Channel 1/Data In 4
//     ComTask Inputs/GVL_COM.stComIn_LAMP_ROUGH_PTM_01/D[5] <-> COM TxPDO-Map Inputs Channel 1/Data In 5
//     ComTask Inputs/GVL_COM.stComIn_LAMP_ROUGH_PTM_01/D[6] <-> COM TxPDO-Map Inputs Channel 1/Data In 6
//     ComTask Inputs/GVL_COM.stComIn_LAMP_ROUGH_PTM_01/D[7] <-> COM TxPDO-Map Inputs Channel 1/Data In 7
//     ComTask Inputs/GVL_COM.stComIn_LAMP_ROUGH_PTM_01/D[8] <-> COM TxPDO-Map Inputs Channel 1/Data In 8
//     ComTask Inputs/GVL_COM.stComIn_LAMP_ROUGH_PTM_01/D[9] <-> COM TxPDO-Map Inputs Channel 1/Data In 9
//     ComTask Inputs/GVL_COM.stComIn_LAMP_ROUGH_PTM_01/Status <-> COM TxPDO-Map Inputs Channel 1/Status
//     ComTask Outputs/GVL_COM.stComOut_LAMP_C1_PTM_01/Ctrl <-> COM RxPDO-Map Outputs Channel 2/Ctrl
//     ComTask Outputs/GVL_COM.stComOut_LAMP_C1_PTM_01/D[0] <-> COM RxPDO-Map Outputs Channel 2/Data Out 0
//     ComTask Outputs/GVL_COM.stComOut_LAMP_C1_PTM_01/D[10] <-> COM RxPDO-Map Outputs Channel 2/Data Out 10
//     ComTask Outputs/GVL_COM.stComOut_LAMP_C1_PTM_01/D[11] <-> COM RxPDO-Map Outputs Channel 2/Data Out 11
//     ComTask Outputs/GVL_COM.stComOut_LAMP_C1_PTM_01/D[12] <-> COM RxPDO-Map Outputs Channel 2/Data Out 12
//     ComTask Outputs/GVL_COM.stComOut_LAMP_C1_PTM_01/D[13] <-> COM RxPDO-Map Outputs Channel 2/Data Out 13
//     ComTask Outputs/GVL_COM.stComOut_LAMP_C1_PTM_01/D[14] <-> COM RxPDO-Map Outputs Channel 2/Data Out 14
//     ComTask Outputs/GVL_COM.stComOut_LAMP_C1_PTM_01/D[15] <-> COM RxPDO-Map Outputs Channel 2/Data Out 15
//     ComTask Outputs/GVL_COM.stComOut_LAMP_C1_PTM_01/D[16] <-> COM RxPDO-Map Outputs Channel 2/Data Out 16
//     ComTask Outputs/GVL_COM.stComOut_LAMP_C1_PTM_01/D[17] <-> COM RxPDO-Map Outputs Channel 2/Data Out 17
//     ComTask Outputs/GVL_COM.stComOut_LAMP_C1_PTM_01/D[18] <-> COM RxPDO-Map Outputs Channel 2/Data Out 18
//     ComTask Outputs/GVL_COM.stComOut_LAMP_C1_PTM_01/D[19] <-> COM RxPDO-Map Outputs Channel 2/Data Out 19
//     ComTask Outputs/GVL_COM.stComOut_LAMP_C1_PTM_01/D[1] <-> COM RxPDO-Map Outputs Channel 2/Data Out 1
//     ComTask Outputs/GVL_COM.stComOut_LAMP_C1_PTM_01/D[20] <-> COM RxPDO-Map Outputs Channel 2/Data Out 20
//     ComTask Outputs/GVL_COM.stComOut_LAMP_C1_PTM_01/D[21] <-> COM RxPDO-Map Outputs Channel 2/Data Out 21
//     ComTask Outputs/GVL_COM.stComOut_LAMP_C1_PTM_01/D[2] <-> COM RxPDO-Map Outputs Channel 2/Data Out 2
//     ComTask Outputs/GVL_COM.stComOut_LAMP_C1_PTM_01/D[3] <-> COM RxPDO-Map Outputs Channel 2/Data Out 3
//     ComTask Outputs/GVL_COM.stComOut_LAMP_C1_PTM_01/D[4] <-> COM RxPDO-Map Outputs Channel 2/Data Out 4
//     ComTask Outputs/GVL_COM.stComOut_LAMP_C1_PTM_01/D[5] <-> COM RxPDO-Map Outputs Channel 2/Data Out 5
//     ComTask Outputs/GVL_COM.stComOut_LAMP_C1_PTM_01/D[6] <-> COM RxPDO-Map Outputs Channel 2/Data Out 6
//     ComTask Outputs/GVL_COM.stComOut_LAMP_C1_PTM_01/D[7] <-> COM RxPDO-Map Outputs Channel 2/Data Out 7
//     ComTask Outputs/GVL_COM.stComOut_LAMP_C1_PTM_01/D[8] <-> COM RxPDO-Map Outputs Channel 2/Data Out 8
//     ComTask Outputs/GVL_COM.stComOut_LAMP_C1_PTM_01/D[9] <-> COM RxPDO-Map Outputs Channel 2/Data Out 9
//     ComTask Outputs/GVL_COM.stComOut_LAMP_ROUGH_PTM_01/Ctrl <-> COM RxPDO-Map Outputs Channel 1/Ctrl
//     ComTask Outputs/GVL_COM.stComOut_LAMP_ROUGH_PTM_01/D[0] <-> COM RxPDO-Map Outputs Channel 1/Data Out 0
//     ComTask Outputs/GVL_COM.stComOut_LAMP_ROUGH_PTM_01/D[10] <-> COM RxPDO-Map Outputs Channel 1/Data Out 10
//     ComTask Outputs/GVL_COM.stComOut_LAMP_ROUGH_PTM_01/D[11] <-> COM RxPDO-Map Outputs Channel 1/Data Out 11
//     ComTask Outputs/GVL_COM.stComOut_LAMP_ROUGH_PTM_01/D[12] <-> COM RxPDO-Map Outputs Channel 1/Data Out 12
//     ComTask Outputs/GVL_COM.stComOut_LAMP_ROUGH_PTM_01/D[13] <-> COM RxPDO-Map Outputs Channel 1/Data Out 13
//     ComTask Outputs/GVL_COM.stComOut_LAMP_ROUGH_PTM_01/D[14] <-> COM RxPDO-Map Outputs Channel 1/Data Out 14
//     ComTask Outputs/GVL_COM.stComOut_LAMP_ROUGH_PTM_01/D[15] <-> COM RxPDO-Map Outputs Channel 1/Data Out 15
//     ComTask Outputs/GVL_COM.stComOut_LAMP_ROUGH_PTM_01/D[16] <-> COM RxPDO-Map Outputs Channel 1/Data Out 16
//     ComTask Outputs/GVL_COM.stComOut_LAMP_ROUGH_PTM_01/D[17] <-> COM RxPDO-Map Outputs Channel 1/Data Out 17
//     ComTask Outputs/GVL_COM.stComOut_LAMP_ROUGH_PTM_01/D[18] <-> COM RxPDO-Map Outputs Channel 1/Data Out 18
//     ComTask Outputs/GVL_COM.stComOut_LAMP_ROUGH_PTM_01/D[19] <-> COM RxPDO-Map Outputs Channel 1/Data Out 19
//     ComTask Outputs/GVL_COM.stComOut_LAMP_ROUGH_PTM_01/D[1] <-> COM RxPDO-Map Outputs Channel 1/Data Out 1
//     ComTask Outputs/GVL_COM.stComOut_LAMP_ROUGH_PTM_01/D[20] <-> COM RxPDO-Map Outputs Channel 1/Data Out 20
//     ComTask Outputs/GVL_COM.stComOut_LAMP_ROUGH_PTM_01/D[21] <-> COM RxPDO-Map Outputs Channel 1/Data Out 21
//     ComTask Outputs/GVL_COM.stComOut_LAMP_ROUGH_PTM_01/D[2] <-> COM RxPDO-Map Outputs Channel 1/Data Out 2
//     ComTask Outputs/GVL_COM.stComOut_LAMP_ROUGH_PTM_01/D[3] <-> COM RxPDO-Map Outputs Channel 1/Data Out 3
//     ComTask Outputs/GVL_COM.stComOut_LAMP_ROUGH_PTM_01/D[4] <-> COM RxPDO-Map Outputs Channel 1/Data Out 4
//     ComTask Outputs/GVL_COM.stComOut_LAMP_ROUGH_PTM_01/D[5] <-> COM RxPDO-Map Outputs Channel 1/Data Out 5
//     ComTask Outputs/GVL_COM.stComOut_LAMP_ROUGH_PTM_01/D[6] <-> COM RxPDO-Map Outputs Channel 1/Data Out 6
//     ComTask Outputs/GVL_COM.stComOut_LAMP_ROUGH_PTM_01/D[7] <-> COM RxPDO-Map Outputs Channel 1/Data Out 7
//     ComTask Outputs/GVL_COM.stComOut_LAMP_ROUGH_PTM_01/D[8] <-> COM RxPDO-Map Outputs Channel 1/Data Out 8
//     ComTask Outputs/GVL_COM.stComOut_LAMP_ROUGH_PTM_01/D[9] <-> COM RxPDO-Map Outputs Channel 1/Data Out 9
//   plc_lamp_lv17_vac/plc_lamp_lv17_vac Instance <-> Device 1 (EtherCAT)/LAMP_PLC_E0_EK1200/LAMP_PLC_E12_EK1122/LAMP_PNL_EP00_EP9128-0021/LAMP_PNL2_EP16_EP2338-0002
//     PlcTask Inputs/GVL_Devices.LAMP_CATCH_PTM_01.i_xAtSpd <-> Channel 1/Input
//     PlcTask Inputs/GVL_Devices.LAMP_CATCH_PTM_02.i_xAtSpd <-> Channel 5/Input
//     PlcTask Inputs/GVL_Devices.LAMP_CATCH_PTM_01.i_xFaultNC <-> Channel 2/Input
//     PlcTask Inputs/GVL_Devices.LAMP_CATCH_PTM_02.i_xFaultNC <-> Channel 6/Input
//   plc_lamp_lv17_vac/plc_lamp_lv17_vac Instance <-> Device 1 (EtherCAT)/LAMP_PLC_E0_EK1200/LAMP_PLC_E12_EK1122/LAMP_PNL_EP00_EP9128-0021/LAMP_PNL2_EP17_EP2624-0002
//     PlcTask Outputs/GVL_Devices.LAMP_CATCH_PTM_01.q_RunDO <-> Channel 1/Output
//     PlcTask Outputs/GVL_Devices.LAMP_CATCH_PTM_02.q_RunDO <-> Channel 3/Output
//     PlcTask Outputs/GVL_Devices.LAMP_CATCH_PTM_01.q_xReset <-> Channel 2/Output
//     PlcTask Outputs/GVL_Devices.LAMP_CATCH_PTM_02.q_xReset <-> Channel 4/Output
//   plc_lamp_lv17_vac/plc_lamp_lv17_vac Instance <-> Device 1 (EtherCAT)/LAMP_PLC_E0_EK1200/LAMP_PLC_E12_EK1122/LAMP_PNL_EP00_EP9128-0021/LAMP_PNL2_EP19_EP3174-0002
//     PlcTask Inputs/GVL_Devices.LAMP_C2_GPI_01.i_iPRESS_R <-> AI Standard Channel 1/Value
//     PlcTask Inputs/GVL_Devices.LAMP_GJ1_GPI_01.i_iPRESS_R <-> AI Standard Channel 3/Value
//     PlcTask Inputs/GVL_Devices.LAMP_GJ2_GPI_01.i_iPRESS_R <-> AI Standard Channel 4/Value
//   plc_lamp_lv17_vac/plc_lamp_lv17_vac Instance <-> Device 1 (EtherCAT)/LAMP_PLC_E0_EK1200/LAMP_PLC_E12_EK1122/LAMP_PNL_EP00_EP9128-0021/LAMP_PNL2_EP20_EP3174-0002
//     PlcTask Inputs/GVL_Devices.LAMP_ROUGH_GPI_01.i_iPRESS_R <-> AI Standard Channel 1/Value
//     PlcTask Inputs/GVL_Devices.LAMP_ROUGH_GPI_02.i_iPRESS_R <-> AI Standard Channel 2/Value
//     PlcTask Inputs/GVL_Devices.LAMP_ROUGH_GPI_03.i_iPRESS_R <-> AI Standard Channel 3/Value
//     PlcTask Inputs/GVL_Devices.LAMP_ROUGH_GPI_04.i_iPRESS_R <-> AI Standard Channel 4/Value
//   plc_lamp_lv17_vac/plc_lamp_lv17_vac Instance <-> Device 1 (EtherCAT)/LAMP_PLC_E0_EK1200/LAMP_PLC_E12_EK1122/LAMP_PNL_EP00_EP9128-0021/LAMP_PNL2_EP21_EP3174-0002
//     PlcTask Inputs/GVL_Devices.LAMP_C2_GCC_01.i_iPRESS_R <-> AI Standard Channel 1/Value
//     PlcTask Inputs/GVL_Devices.LAMP_CATCH_GCC_01.i_iPRESS_R <-> AI Standard Channel 2/Value
//     PlcTask Inputs/GVL_Devices.LAMP_CATCH_GCC_02.i_iPRESS_R <-> AI Standard Channel 3/Value
//     PlcTask Inputs/GVL_Devices.LAMP_GJ1_GCC_01.i_iPRESS_R <-> AI Standard Channel 4/Value
//   plc_lamp_lv17_vac/plc_lamp_lv17_vac Instance <-> Device 1 (EtherCAT)/LAMP_PLC_E0_EK1200/LAMP_PLC_E12_EK1122/LAMP_PNL_EP00_EP9128-0021/LAMP_PNL2_EP22_EP2624-0002
//     PlcTask Outputs/GVL_Devices.LAMP_C2_GCC_01.q_xHV_DIS <-> Channel 1/Output
//     PlcTask Outputs/GVL_Devices.LAMP_CATCH_GCC_01.q_xHV_DIS <-> Channel 2/Output
//     PlcTask Outputs/GVL_Devices.LAMP_CATCH_GCC_02.q_xHV_DIS <-> Channel 3/Output
//     PlcTask Outputs/GVL_Devices.LAMP_GJ1_GCC_01.q_xHV_DIS <-> Channel 4/Output
//   plc_lamp_lv17_vac/plc_lamp_lv17_vac Instance <-> Device 1 (EtherCAT)/LAMP_PLC_E0_EK1200/LAMP_PLC_E12_EK1122/LAMP_PNL_EP00_EP9128-0021/LAMP_PNL2_EP23_EP3174-0002
//     PlcTask Inputs/GVL_Devices.LAMP_C1_GHC_01.i_iPRESS_R <-> AI Standard Channel 2/Value
//     PlcTask Inputs/GVL_Devices.LAMP_GJ2_GCC_01.i_iPRESS_R <-> AI Standard Channel 1/Value
//   plc_lamp_lv17_vac/plc_lamp_lv17_vac Instance <-> Device 1 (EtherCAT)/LAMP_PLC_E0_EK1200/LAMP_PLC_E12_EK1122/LAMP_PNL_EP00_EP9128-0021/LAMP_PNL2_EP24_EP2624-0002
//     PlcTask Outputs/GVL_Devices.LAMP_C1_GHC_01.q_xHV_DIS <-> Channel 2/Output
//     PlcTask Outputs/GVL_Devices.LAMP_GJ2_GCC_01.q_xHV_DIS <-> Channel 1/Output
//   plc_lamp_lv17_vac/plc_lamp_lv17_vac Instance <-> Device 1 (EtherCAT)/LAMP_PLC_E0_EK1200/LAMP_PLC_E12_EK1122/LAMP_PNL_EP00_EP9128-0021/LAMP_PNL2_EP25_EP2338-0002
//     PlcTask Inputs/GVL_Devices.LAMP_ROUGH_VRC_01.i_xClsLS <-> Channel 2/Input
//     PlcTask Inputs/GVL_Devices.LAMP_ROUGH_VRC_02.i_xClsLS <-> Channel 6/Input
//     PlcTask Inputs/GVL_Devices.LAMP_ROUGH_VRC_01.i_xOpnLS <-> Channel 1/Input
//     PlcTask Inputs/GVL_Devices.LAMP_ROUGH_VRC_02.i_xOpnLS <-> Channel 5/Input
//     PlcTask Outputs/GVL_Devices.LAMP_ROUGH_VRC_01.q_xOPN_DO <-> Channel 11/Output
//     PlcTask Outputs/GVL_Devices.LAMP_ROUGH_VRC_02.q_xCLS_DO <-> Channel 15/Output
//   plc_lamp_lv17_vac/plc_lamp_lv17_vac Instance <-> Device 1 (EtherCAT)/LAMP_PLC_E0_EK1200/LAMP_PLC_E12_EK1122/LAMP_PNL_EP00_EP9128-0021/LAMP_PNL2_EP26_EP2338-0002
//     PlcTask Inputs/GVL_Devices.LAMP_ROUGH_VRC_03.i_xClsLS <-> Channel 2/Input
//     PlcTask Inputs/GVL_Devices.LAMP_ROUGH_VRC_03.i_xOpnLS <-> Channel 1/Input
//     PlcTask Outputs/GVL_Devices.LAMP_ROUGH_VRC_03.q_xOPN_DO <-> Channel 11/Output
//   plc_lamp_lv17_vac/plc_lamp_lv17_vac Instance <-> Device 1 (EtherCAT)/LAMP_PLC_E0_EK1200/LAMP_PLC_E12_EK1122/LAMP_PNL_EP00_EP9128-0021/Term 88 (EP9128-1021)/LAMP_CLSTR1_PNL1_EP01_EP2338-0002
//     PlcTask Inputs/GVL_Devices.LAMP_CLSTR1_PTM_01.i_xAtSpd <-> Channel 1/Input
//     PlcTask Inputs/GVL_Devices.LAMP_CLSTR1_PTM_01.i_xFaultNC <-> Channel 2/Input
//     PlcTask Inputs/GVL_Devices.LAMP_CLSTR1_PTM_01.i_xRemote <-> Channel 3/Input
//   plc_lamp_lv17_vac/plc_lamp_lv17_vac Instance <-> Device 1 (EtherCAT)/LAMP_PLC_E0_EK1200/LAMP_PLC_E12_EK1122/LAMP_PNL_EP00_EP9128-0021/Term 88 (EP9128-1021)/LAMP_CLSTR1_PNL1_EP03_EP6002-0002
//     ComTask Inputs/GVL_COM.stComIn_LAMP_CLSTR1_PTM_01/D[0] <-> COM TxPDO-Map Inputs Channel 1/Data In 0
//     ComTask Inputs/GVL_COM.stComIn_LAMP_CLSTR1_PTM_01/D[10] <-> COM TxPDO-Map Inputs Channel 1/Data In 10
//     ComTask Inputs/GVL_COM.stComIn_LAMP_CLSTR1_PTM_01/D[11] <-> COM TxPDO-Map Inputs Channel 1/Data In 11
//     ComTask Inputs/GVL_COM.stComIn_LAMP_CLSTR1_PTM_01/D[12] <-> COM TxPDO-Map Inputs Channel 1/Data In 12
//     ComTask Inputs/GVL_COM.stComIn_LAMP_CLSTR1_PTM_01/D[13] <-> COM TxPDO-Map Inputs Channel 1/Data In 13
//     ComTask Inputs/GVL_COM.stComIn_LAMP_CLSTR1_PTM_01/D[14] <-> COM TxPDO-Map Inputs Channel 1/Data In 14
//     ComTask Inputs/GVL_COM.stComIn_LAMP_CLSTR1_PTM_01/D[15] <-> COM TxPDO-Map Inputs Channel 1/Data In 15
//     ComTask Inputs/GVL_COM.stComIn_LAMP_CLSTR1_PTM_01/D[16] <-> COM TxPDO-Map Inputs Channel 1/Data In 16
//     ComTask Inputs/GVL_COM.stComIn_LAMP_CLSTR1_PTM_01/D[17] <-> COM TxPDO-Map Inputs Channel 1/Data In 17
//     ComTask Inputs/GVL_COM.stComIn_LAMP_CLSTR1_PTM_01/D[18] <-> COM TxPDO-Map Inputs Channel 1/Data In 18
//     ComTask Inputs/GVL_COM.stComIn_LAMP_CLSTR1_PTM_01/D[19] <-> COM TxPDO-Map Inputs Channel 1/Data In 19
//     ComTask Inputs/GVL_COM.stComIn_LAMP_CLSTR1_PTM_01/D[1] <-> COM TxPDO-Map Inputs Channel 1/Data In 1
//     ComTask Inputs/GVL_COM.stComIn_LAMP_CLSTR1_PTM_01/D[20] <-> COM TxPDO-Map Inputs Channel 1/Data In 20
//     ComTask Inputs/GVL_COM.stComIn_LAMP_CLSTR1_PTM_01/D[21] <-> COM TxPDO-Map Inputs Channel 1/Data In 21
//     ComTask Inputs/GVL_COM.stComIn_LAMP_CLSTR1_PTM_01/D[2] <-> COM TxPDO-Map Inputs Channel 1/Data In 2
//     ComTask Inputs/GVL_COM.stComIn_LAMP_CLSTR1_PTM_01/D[3] <-> COM TxPDO-Map Inputs Channel 1/Data In 3
//     ComTask Inputs/GVL_COM.stComIn_LAMP_CLSTR1_PTM_01/D[4] <-> COM TxPDO-Map Inputs Channel 1/Data In 4
//     ComTask Inputs/GVL_COM.stComIn_LAMP_CLSTR1_PTM_01/D[5] <-> COM TxPDO-Map Inputs Channel 1/Data In 5
//     ComTask Inputs/GVL_COM.stComIn_LAMP_CLSTR1_PTM_01/D[6] <-> COM TxPDO-Map Inputs Channel 1/Data In 6
//     ComTask Inputs/GVL_COM.stComIn_LAMP_CLSTR1_PTM_01/D[7] <-> COM TxPDO-Map Inputs Channel 1/Data In 7
//     ComTask Inputs/GVL_COM.stComIn_LAMP_CLSTR1_PTM_01/D[8] <-> COM TxPDO-Map Inputs Channel 1/Data In 8
//     ComTask Inputs/GVL_COM.stComIn_LAMP_CLSTR1_PTM_01/D[9] <-> COM TxPDO-Map Inputs Channel 1/Data In 9
//     ComTask Inputs/GVL_COM.stComIn_LAMP_CLSTR1_PTM_01/Status <-> COM TxPDO-Map Inputs Channel 1/Status
//     ComTask Outputs/GVL_COM.stComOut_LAMP_CLSTR1_PTM_01/Ctrl <-> COM RxPDO-Map Outputs Channel 1/Ctrl
//     ComTask Outputs/GVL_COM.stComOut_LAMP_CLSTR1_PTM_01/D[0] <-> COM RxPDO-Map Outputs Channel 1/Data Out 0
//     ComTask Outputs/GVL_COM.stComOut_LAMP_CLSTR1_PTM_01/D[10] <-> COM RxPDO-Map Outputs Channel 1/Data Out 10
//     ComTask Outputs/GVL_COM.stComOut_LAMP_CLSTR1_PTM_01/D[11] <-> COM RxPDO-Map Outputs Channel 1/Data Out 11
//     ComTask Outputs/GVL_COM.stComOut_LAMP_CLSTR1_PTM_01/D[12] <-> COM RxPDO-Map Outputs Channel 1/Data Out 12
//     ComTask Outputs/GVL_COM.stComOut_LAMP_CLSTR1_PTM_01/D[13] <-> COM RxPDO-Map Outputs Channel 1/Data Out 13
//     ComTask Outputs/GVL_COM.stComOut_LAMP_CLSTR1_PTM_01/D[14] <-> COM RxPDO-Map Outputs Channel 1/Data Out 14
//     ComTask Outputs/GVL_COM.stComOut_LAMP_CLSTR1_PTM_01/D[15] <-> COM RxPDO-Map Outputs Channel 1/Data Out 15
//     ComTask Outputs/GVL_COM.stComOut_LAMP_CLSTR1_PTM_01/D[16] <-> COM RxPDO-Map Outputs Channel 1/Data Out 16
//     ComTask Outputs/GVL_COM.stComOut_LAMP_CLSTR1_PTM_01/D[17] <-> COM RxPDO-Map Outputs Channel 1/Data Out 17
//     ComTask Outputs/GVL_COM.stComOut_LAMP_CLSTR1_PTM_01/D[18] <-> COM RxPDO-Map Outputs Channel 1/Data Out 18
//     ComTask Outputs/GVL_COM.stComOut_LAMP_CLSTR1_PTM_01/D[19] <-> COM RxPDO-Map Outputs Channel 1/Data Out 19
//     ComTask Outputs/GVL_COM.stComOut_LAMP_CLSTR1_PTM_01/D[1] <-> COM RxPDO-Map Outputs Channel 1/Data Out 1
//     ComTask Outputs/GVL_COM.stComOut_LAMP_CLSTR1_PTM_01/D[20] <-> COM RxPDO-Map Outputs Channel 1/Data Out 20
//     ComTask Outputs/GVL_COM.stComOut_LAMP_CLSTR1_PTM_01/D[21] <-> COM RxPDO-Map Outputs Channel 1/Data Out 21
//     ComTask Outputs/GVL_COM.stComOut_LAMP_CLSTR1_PTM_01/D[2] <-> COM RxPDO-Map Outputs Channel 1/Data Out 2
//     ComTask Outputs/GVL_COM.stComOut_LAMP_CLSTR1_PTM_01/D[3] <-> COM RxPDO-Map Outputs Channel 1/Data Out 3
//     ComTask Outputs/GVL_COM.stComOut_LAMP_CLSTR1_PTM_01/D[4] <-> COM RxPDO-Map Outputs Channel 1/Data Out 4
//     ComTask Outputs/GVL_COM.stComOut_LAMP_CLSTR1_PTM_01/D[5] <-> COM RxPDO-Map Outputs Channel 1/Data Out 5
//     ComTask Outputs/GVL_COM.stComOut_LAMP_CLSTR1_PTM_01/D[6] <-> COM RxPDO-Map Outputs Channel 1/Data Out 6
//     ComTask Outputs/GVL_COM.stComOut_LAMP_CLSTR1_PTM_01/D[7] <-> COM RxPDO-Map Outputs Channel 1/Data Out 7
//     ComTask Outputs/GVL_COM.stComOut_LAMP_CLSTR1_PTM_01/D[8] <-> COM RxPDO-Map Outputs Channel 1/Data Out 8
//     ComTask Outputs/GVL_COM.stComOut_LAMP_CLSTR1_PTM_01/D[9] <-> COM RxPDO-Map Outputs Channel 1/Data Out 9
//   plc_lamp_lv17_vac/plc_lamp_lv17_vac Instance <-> Device 1 (EtherCAT)/LAMP_PLC_E0_EK1200/LAMP_PLC_E12_EK1122/LAMP_PNL_EP00_EP9128-0021/Term 88 (EP9128-1021)/LAMP_CLSTR1_PNL3_EP01_EP2338-0002
//     PlcTask Inputs/GVL_Devices.LAMP_CLSTR1_PTM_03.i_xAtSpd <-> Channel 1/Input
//     PlcTask Inputs/GVL_Devices.LAMP_CLSTR1_PTM_03.i_xFaultNC <-> Channel 2/Input
//     PlcTask Inputs/GVL_Devices.LAMP_CLSTR1_PTM_03.i_xRemote <-> Channel 3/Input
//   plc_lamp_lv17_vac/plc_lamp_lv17_vac Instance <-> Device 1 (EtherCAT)/LAMP_PLC_E0_EK1200/LAMP_PLC_E12_EK1122/LAMP_PNL_EP00_EP9128-0021/Term 88 (EP9128-1021)/LAMP_CLSTR1_PNL3_EP02_EP2624-0002
//     PlcTask Outputs/GVL_Devices.LAMP_CLSTR1_PTM_03.q_RunDO <-> Channel 1/Output
//     PlcTask Outputs/GVL_Devices.LAMP_CLSTR1_PTM_03.q_xReset <-> Channel 2/Output
//   plc_lamp_lv17_vac/plc_lamp_lv17_vac Instance <-> Device 1 (EtherCAT)/LAMP_PLC_E0_EK1200/LAMP_PLC_E12_EK1122/LAMP_PNL_EP00_EP9128-0021/Term 88 (EP9128-1021)/LAMP_CLSTR1_PNL3_EP03_EP6002-0002
//     ComTask Inputs/GVL_COM.stComIn_LAMP_CLSTR1_PTM_03/D[0] <-> COM TxPDO-Map Inputs Channel 1/Data In 0
//     ComTask Inputs/GVL_COM.stComIn_LAMP_CLSTR1_PTM_03/D[10] <-> COM TxPDO-Map Inputs Channel 1/Data In 10
//     ComTask Inputs/GVL_COM.stComIn_LAMP_CLSTR1_PTM_03/D[11] <-> COM TxPDO-Map Inputs Channel 1/Data In 11
//     ComTask Inputs/GVL_COM.stComIn_LAMP_CLSTR1_PTM_03/D[12] <-> COM TxPDO-Map Inputs Channel 1/Data In 12
//     ComTask Inputs/GVL_COM.stComIn_LAMP_CLSTR1_PTM_03/D[13] <-> COM TxPDO-Map Inputs Channel 1/Data In 13
//     ComTask Inputs/GVL_COM.stComIn_LAMP_CLSTR1_PTM_03/D[14] <-> COM TxPDO-Map Inputs Channel 1/Data In 14
//     ComTask Inputs/GVL_COM.stComIn_LAMP_CLSTR1_PTM_03/D[15] <-> COM TxPDO-Map Inputs Channel 1/Data In 15
//     ComTask Inputs/GVL_COM.stComIn_LAMP_CLSTR1_PTM_03/D[16] <-> COM TxPDO-Map Inputs Channel 1/Data In 16
//     ComTask Inputs/GVL_COM.stComIn_LAMP_CLSTR1_PTM_03/D[17] <-> COM TxPDO-Map Inputs Channel 1/Data In 17
//     ComTask Inputs/GVL_COM.stComIn_LAMP_CLSTR1_PTM_03/D[18] <-> COM TxPDO-Map Inputs Channel 1/Data In 18
//     ComTask Inputs/GVL_COM.stComIn_LAMP_CLSTR1_PTM_03/D[19] <-> COM TxPDO-Map Inputs Channel 1/Data In 19
//     ComTask Inputs/GVL_COM.stComIn_LAMP_CLSTR1_PTM_03/D[1] <-> COM TxPDO-Map Inputs Channel 1/Data In 1
//     ComTask Inputs/GVL_COM.stComIn_LAMP_CLSTR1_PTM_03/D[20] <-> COM TxPDO-Map Inputs Channel 1/Data In 20
//     ComTask Inputs/GVL_COM.stComIn_LAMP_CLSTR1_PTM_03/D[21] <-> COM TxPDO-Map Inputs Channel 1/Data In 21
//     ComTask Inputs/GVL_COM.stComIn_LAMP_CLSTR1_PTM_03/D[2] <-> COM TxPDO-Map Inputs Channel 1/Data In 2
//     ComTask Inputs/GVL_COM.stComIn_LAMP_CLSTR1_PTM_03/D[3] <-> COM TxPDO-Map Inputs Channel 1/Data In 3
//     ComTask Inputs/GVL_COM.stComIn_LAMP_CLSTR1_PTM_03/D[4] <-> COM TxPDO-Map Inputs Channel 1/Data In 4
//     ComTask Inputs/GVL_COM.stComIn_LAMP_CLSTR1_PTM_03/D[5] <-> COM TxPDO-Map Inputs Channel 1/Data In 5
//     ComTask Inputs/GVL_COM.stComIn_LAMP_CLSTR1_PTM_03/D[6] <-> COM TxPDO-Map Inputs Channel 1/Data In 6
//     ComTask Inputs/GVL_COM.stComIn_LAMP_CLSTR1_PTM_03/D[7] <-> COM TxPDO-Map Inputs Channel 1/Data In 7
//     ComTask Inputs/GVL_COM.stComIn_LAMP_CLSTR1_PTM_03/D[8] <-> COM TxPDO-Map Inputs Channel 1/Data In 8
//     ComTask Inputs/GVL_COM.stComIn_LAMP_CLSTR1_PTM_03/D[9] <-> COM TxPDO-Map Inputs Channel 1/Data In 9
//     ComTask Inputs/GVL_COM.stComIn_LAMP_CLSTR1_PTM_03/Status <-> COM TxPDO-Map Inputs Channel 1/Status
//     ComTask Outputs/GVL_COM.stComOut_LAMP_CLSTR1_PTM_03/Ctrl <-> COM RxPDO-Map Outputs Channel 1/Ctrl
//     ComTask Outputs/GVL_COM.stComOut_LAMP_CLSTR1_PTM_03/D[0] <-> COM RxPDO-Map Outputs Channel 1/Data Out 0
//     ComTask Outputs/GVL_COM.stComOut_LAMP_CLSTR1_PTM_03/D[10] <-> COM RxPDO-Map Outputs Channel 1/Data Out 10
//     ComTask Outputs/GVL_COM.stComOut_LAMP_CLSTR1_PTM_03/D[11] <-> COM RxPDO-Map Outputs Channel 1/Data Out 11
//     ComTask Outputs/GVL_COM.stComOut_LAMP_CLSTR1_PTM_03/D[12] <-> COM RxPDO-Map Outputs Channel 1/Data Out 12
//     ComTask Outputs/GVL_COM.stComOut_LAMP_CLSTR1_PTM_03/D[13] <-> COM RxPDO-Map Outputs Channel 1/Data Out 13
//     ComTask Outputs/GVL_COM.stComOut_LAMP_CLSTR1_PTM_03/D[14] <-> COM RxPDO-Map Outputs Channel 1/Data Out 14
//     ComTask Outputs/GVL_COM.stComOut_LAMP_CLSTR1_PTM_03/D[15] <-> COM RxPDO-Map Outputs Channel 1/Data Out 15
//     ComTask Outputs/GVL_COM.stComOut_LAMP_CLSTR1_PTM_03/D[16] <-> COM RxPDO-Map Outputs Channel 1/Data Out 16
//     ComTask Outputs/GVL_COM.stComOut_LAMP_CLSTR1_PTM_03/D[17] <-> COM RxPDO-Map Outputs Channel 1/Data Out 17
//     ComTask Outputs/GVL_COM.stComOut_LAMP_CLSTR1_PTM_03/D[18] <-> COM RxPDO-Map Outputs Channel 1/Data Out 18
//     ComTask Outputs/GVL_COM.stComOut_LAMP_CLSTR1_PTM_03/D[19] <-> COM RxPDO-Map Outputs Channel 1/Data Out 19
//     ComTask Outputs/GVL_COM.stComOut_LAMP_CLSTR1_PTM_03/D[1] <-> COM RxPDO-Map Outputs Channel 1/Data Out 1
//     ComTask Outputs/GVL_COM.stComOut_LAMP_CLSTR1_PTM_03/D[20] <-> COM RxPDO-Map Outputs Channel 1/Data Out 20
//     ComTask Outputs/GVL_COM.stComOut_LAMP_CLSTR1_PTM_03/D[21] <-> COM RxPDO-Map Outputs Channel 1/Data Out 21
//     ComTask Outputs/GVL_COM.stComOut_LAMP_CLSTR1_PTM_03/D[2] <-> COM RxPDO-Map Outputs Channel 1/Data Out 2
//     ComTask Outputs/GVL_COM.stComOut_LAMP_CLSTR1_PTM_03/D[3] <-> COM RxPDO-Map Outputs Channel 1/Data Out 3
//     ComTask Outputs/GVL_COM.stComOut_LAMP_CLSTR1_PTM_03/D[4] <-> COM RxPDO-Map Outputs Channel 1/Data Out 4
//     ComTask Outputs/GVL_COM.stComOut_LAMP_CLSTR1_PTM_03/D[5] <-> COM RxPDO-Map Outputs Channel 1/Data Out 5
//     ComTask Outputs/GVL_COM.stComOut_LAMP_CLSTR1_PTM_03/D[6] <-> COM RxPDO-Map Outputs Channel 1/Data Out 6
//     ComTask Outputs/GVL_COM.stComOut_LAMP_CLSTR1_PTM_03/D[7] <-> COM RxPDO-Map Outputs Channel 1/Data Out 7
//     ComTask Outputs/GVL_COM.stComOut_LAMP_CLSTR1_PTM_03/D[8] <-> COM RxPDO-Map Outputs Channel 1/Data Out 8
//     ComTask Outputs/GVL_COM.stComOut_LAMP_CLSTR1_PTM_03/D[9] <-> COM RxPDO-Map Outputs Channel 1/Data Out 9
//   plc_lamp_lv17_vac/plc_lamp_lv17_vac Instance <-> Device 1 (EtherCAT)/LAMP_PLC_E0_EK1200/LAMP_PLC_E12_EK1122/LAMP_PNL_EP00_EP9128-0021/Term 89 (EP9128-2021)/LAMP_CLSTR1_PNL2_EP01_EP2338-0002
//     PlcTask Inputs/GVL_Devices.LAMP_CLSTR1_PTM_02.i_xAtSpd <-> Channel 1/Input
//     PlcTask Inputs/GVL_Devices.LAMP_CLSTR1_PTM_02.i_xFaultNC <-> Channel 2/Input
//     PlcTask Inputs/GVL_Devices.LAMP_CLSTR1_PTM_02.i_xRemote <-> Channel 3/Input
//   plc_lamp_lv17_vac/plc_lamp_lv17_vac Instance <-> Device 1 (EtherCAT)/LAMP_PLC_E0_EK1200/LAMP_PLC_E12_EK1122/LAMP_PNL_EP00_EP9128-0021/Term 89 (EP9128-2021)/LAMP_CLSTR1_PNL2_EP02_EP2624-0002
//     PlcTask Outputs/GVL_Devices.LAMP_CLSTR1_PTM_02.q_RunDO <-> Channel 1/Output
//     PlcTask Outputs/GVL_Devices.LAMP_CLSTR1_PTM_02.q_xReset <-> Channel 2/Output
//   plc_lamp_lv17_vac/plc_lamp_lv17_vac Instance <-> Device 1 (EtherCAT)/LAMP_PLC_E0_EK1200/LAMP_PLC_E12_EK1122/LAMP_PNL_EP00_EP9128-0021/Term 89 (EP9128-2021)/LAMP_CLSTR1_PNL2_EP03_EP6002-0002
//     ComTask Inputs/GVL_COM.stComIn_LAMP_CLSTR1_PTM_02/D[0] <-> COM TxPDO-Map Inputs Channel 1/Data In 0
//     ComTask Inputs/GVL_COM.stComIn_LAMP_CLSTR1_PTM_02/D[10] <-> COM TxPDO-Map Inputs Channel 1/Data In 10
//     ComTask Inputs/GVL_COM.stComIn_LAMP_CLSTR1_PTM_02/D[11] <-> COM TxPDO-Map Inputs Channel 1/Data In 11
//     ComTask Inputs/GVL_COM.stComIn_LAMP_CLSTR1_PTM_02/D[12] <-> COM TxPDO-Map Inputs Channel 1/Data In 12
//     ComTask Inputs/GVL_COM.stComIn_LAMP_CLSTR1_PTM_02/D[13] <-> COM TxPDO-Map Inputs Channel 1/Data In 13
//     ComTask Inputs/GVL_COM.stComIn_LAMP_CLSTR1_PTM_02/D[14] <-> COM TxPDO-Map Inputs Channel 1/Data In 14
//     ComTask Inputs/GVL_COM.stComIn_LAMP_CLSTR1_PTM_02/D[15] <-> COM TxPDO-Map Inputs Channel 1/Data In 15
//     ComTask Inputs/GVL_COM.stComIn_LAMP_CLSTR1_PTM_02/D[16] <-> COM TxPDO-Map Inputs Channel 1/Data In 16
//     ComTask Inputs/GVL_COM.stComIn_LAMP_CLSTR1_PTM_02/D[17] <-> COM TxPDO-Map Inputs Channel 1/Data In 17
//     ComTask Inputs/GVL_COM.stComIn_LAMP_CLSTR1_PTM_02/D[18] <-> COM TxPDO-Map Inputs Channel 1/Data In 18
//     ComTask Inputs/GVL_COM.stComIn_LAMP_CLSTR1_PTM_02/D[19] <-> COM TxPDO-Map Inputs Channel 1/Data In 19
//     ComTask Inputs/GVL_COM.stComIn_LAMP_CLSTR1_PTM_02/D[1] <-> COM TxPDO-Map Inputs Channel 1/Data In 1
//     ComTask Inputs/GVL_COM.stComIn_LAMP_CLSTR1_PTM_02/D[20] <-> COM TxPDO-Map Inputs Channel 1/Data In 20
//     ComTask Inputs/GVL_COM.stComIn_LAMP_CLSTR1_PTM_02/D[21] <-> COM TxPDO-Map Inputs Channel 1/Data In 21
//     ComTask Inputs/GVL_COM.stComIn_LAMP_CLSTR1_PTM_02/D[2] <-> COM TxPDO-Map Inputs Channel 1/Data In 2
//     ComTask Inputs/GVL_COM.stComIn_LAMP_CLSTR1_PTM_02/D[3] <-> COM TxPDO-Map Inputs Channel 1/Data In 3
//     ComTask Inputs/GVL_COM.stComIn_LAMP_CLSTR1_PTM_02/D[4] <-> COM TxPDO-Map Inputs Channel 1/Data In 4
//     ComTask Inputs/GVL_COM.stComIn_LAMP_CLSTR1_PTM_02/D[5] <-> COM TxPDO-Map Inputs Channel 1/Data In 5
//     ComTask Inputs/GVL_COM.stComIn_LAMP_CLSTR1_PTM_02/D[6] <-> COM TxPDO-Map Inputs Channel 1/Data In 6
//     ComTask Inputs/GVL_COM.stComIn_LAMP_CLSTR1_PTM_02/D[7] <-> COM TxPDO-Map Inputs Channel 1/Data In 7
//     ComTask Inputs/GVL_COM.stComIn_LAMP_CLSTR1_PTM_02/D[8] <-> COM TxPDO-Map Inputs Channel 1/Data In 8
//     ComTask Inputs/GVL_COM.stComIn_LAMP_CLSTR1_PTM_02/D[9] <-> COM TxPDO-Map Inputs Channel 1/Data In 9
//     ComTask Inputs/GVL_COM.stComIn_LAMP_CLSTR1_PTM_02/Status <-> COM TxPDO-Map Inputs Channel 1/Status
//     ComTask Outputs/GVL_COM.stComOut_LAMP_CLSTR1_PTM_02/Ctrl <-> COM RxPDO-Map Outputs Channel 1/Ctrl
//     ComTask Outputs/GVL_COM.stComOut_LAMP_CLSTR1_PTM_02/D[0] <-> COM RxPDO-Map Outputs Channel 1/Data Out 0
//     ComTask Outputs/GVL_COM.stComOut_LAMP_CLSTR1_PTM_02/D[10] <-> COM RxPDO-Map Outputs Channel 1/Data Out 10
//     ComTask Outputs/GVL_COM.stComOut_LAMP_CLSTR1_PTM_02/D[11] <-> COM RxPDO-Map Outputs Channel 1/Data Out 11
//     ComTask Outputs/GVL_COM.stComOut_LAMP_CLSTR1_PTM_02/D[12] <-> COM RxPDO-Map Outputs Channel 1/Data Out 12
//     ComTask Outputs/GVL_COM.stComOut_LAMP_CLSTR1_PTM_02/D[13] <-> COM RxPDO-Map Outputs Channel 1/Data Out 13
//     ComTask Outputs/GVL_COM.stComOut_LAMP_CLSTR1_PTM_02/D[14] <-> COM RxPDO-Map Outputs Channel 1/Data Out 14
//     ComTask Outputs/GVL_COM.stComOut_LAMP_CLSTR1_PTM_02/D[15] <-> COM RxPDO-Map Outputs Channel 1/Data Out 15
//     ComTask Outputs/GVL_COM.stComOut_LAMP_CLSTR1_PTM_02/D[16] <-> COM RxPDO-Map Outputs Channel 1/Data Out 16
//     ComTask Outputs/GVL_COM.stComOut_LAMP_CLSTR1_PTM_02/D[17] <-> COM RxPDO-Map Outputs Channel 1/Data Out 17
//     ComTask Outputs/GVL_COM.stComOut_LAMP_CLSTR1_PTM_02/D[18] <-> COM RxPDO-Map Outputs Channel 1/Data Out 18
//     ComTask Outputs/GVL_COM.stComOut_LAMP_CLSTR1_PTM_02/D[19] <-> COM RxPDO-Map Outputs Channel 1/Data Out 19
//     ComTask Outputs/GVL_COM.stComOut_LAMP_CLSTR1_PTM_02/D[1] <-> COM RxPDO-Map Outputs Channel 1/Data Out 1
//     ComTask Outputs/GVL_COM.stComOut_LAMP_CLSTR1_PTM_02/D[20] <-> COM RxPDO-Map Outputs Channel 1/Data Out 20
//     ComTask Outputs/GVL_COM.stComOut_LAMP_CLSTR1_PTM_02/D[21] <-> COM RxPDO-Map Outputs Channel 1/Data Out 21
//     ComTask Outputs/GVL_COM.stComOut_LAMP_CLSTR1_PTM_02/D[2] <-> COM RxPDO-Map Outputs Channel 1/Data Out 2
//     ComTask Outputs/GVL_COM.stComOut_LAMP_CLSTR1_PTM_02/D[3] <-> COM RxPDO-Map Outputs Channel 1/Data Out 3
//     ComTask Outputs/GVL_COM.stComOut_LAMP_CLSTR1_PTM_02/D[4] <-> COM RxPDO-Map Outputs Channel 1/Data Out 4
//     ComTask Outputs/GVL_COM.stComOut_LAMP_CLSTR1_PTM_02/D[5] <-> COM RxPDO-Map Outputs Channel 1/Data Out 5
//     ComTask Outputs/GVL_COM.stComOut_LAMP_CLSTR1_PTM_02/D[6] <-> COM RxPDO-Map Outputs Channel 1/Data Out 6
//     ComTask Outputs/GVL_COM.stComOut_LAMP_CLSTR1_PTM_02/D[7] <-> COM RxPDO-Map Outputs Channel 1/Data Out 7
//     ComTask Outputs/GVL_COM.stComOut_LAMP_CLSTR1_PTM_02/D[8] <-> COM RxPDO-Map Outputs Channel 1/Data Out 8
//     ComTask Outputs/GVL_COM.stComOut_LAMP_CLSTR1_PTM_02/D[9] <-> COM RxPDO-Map Outputs Channel 1/Data Out 9
//   plc_lamp_lv17_vac/plc_lamp_lv17_vac Instance <-> Device 1 (EtherCAT)/LAMP_PLC_E0_EK1200/LAMP_PLC_E3_EL6692
//     PlcTask Inputs/GVL_PLC_Interfaces.sHUTCH_PLC_NAME <-> IO Inputs/HUTCH_PLC_NAME
//     PlcTask Inputs/GVL_PLC_Interfaces.xEcatBridge_TxPDO_state <-> SYNC Inputs/TxPDO state
//     PlcTask Inputs/GVL_PLC_Interfaces.xEcatBridge_WcState <-> WcState/WcState
//     PlcTask Inputs/GVL_PLC_Interfaces.xTMO_ROUGH1_VRC_01_OPEN_LS <-> IO Inputs/TMO_ROUGH1_VRC_01_OPEN_LS
//     PlcTask Inputs/GVL_PLC_Interfaces.xTMO_ROUGH2_VRC_01_OPEN_LS <-> IO Inputs/TMO_ROUGH2_VRC_01_OPEN_LS
//     PlcTask Outputs/GVL_PLC_Interfaces.rIP1_MAIN_rPRESS <-> IO Outputs/IP1_MAIN_rPRESS
//     PlcTask Outputs/GVL_PLC_Interfaces.sENDSTATION_PLC_NAME <-> IO Outputs/ENDSTATION_PLC_NAME
//     PlcTask Outputs/GVL_PLC_Interfaces.xIP1_HV_SAFETY_ENABLE <-> IO Outputs/IP1_HV_SAFETY_ENABLE
//     PlcTask Outputs/GVL_PLC_Interfaces.xIP1_MAIN_xAT_VAC <-> IO Outputs/IP1_MAIN_xAT_VAC
//     PlcTask Outputs/GVL_PLC_Interfaces.xIP1_MAIN_xPRESS_OK <-> IO Outputs/IP1_MAIN_xPRESS_OK
//     PlcTask Outputs/GVL_PLC_Interfaces.xIP1_ROUGH_VRC_01_OPEN_LS <-> IO Outputs/IP1_ROUGH_VRC_01_OPEN_LS
//     PlcTask Outputs/GVL_PLC_Interfaces.xIP1_ROUGH_VRC_02_OPEN_LS <-> IO Outputs/IP1_ROUGH_VRC_02_OPEN_LS
//     PlcTask Outputs/GVL_PLC_Interfaces.xIP1_ROUGH_VRC_03_OPEN_LS <-> IO Outputs/IP1_ROUGH_VRC_03_OPEN_LS
//     PlcTask Outputs/GVL_PLC_Interfaces.xIP1_TURBOS_ALL_AtSpd <-> IO Outputs/IP1_TURBOS_ALL_AtSpd
//   plc_lamp_lv17_vac/plc_lamp_lv17_vac Instance <-> Device 1 (EtherCAT)/LAMP_PLC_E0_EK1200/LAMP_PLC_E8_EL2794
//     PlcTask Outputs/GVL_PLC_Interfaces.xHighVoltageSafteyLoopEnable <-> Channel 1/Output

// ---- GVLs/GVL_COM.TcGVL
//{attribute 'qualified_only'}
VAR_GLOBAL
// Define COM Ports/Buffers incl. library Tc2_SerialCom
	SerialRXBuffer_LAMP_C2_PTM_01 : ComBuffer;
	SerialTXBuffer_LAMP_C2_PTM_01 : ComBuffer;	
	SerialRXBuffer_LAMP_C2_PTM_02 : ComBuffer;
	SerialTXBuffer_LAMP_C2_PTM_02 : ComBuffer;	
	SerialRXBuffer_LAMP_C2_PTM_03 : ComBuffer;
	SerialTXBuffer_LAMP_C2_PTM_03 : ComBuffer;	
	SerialRXBuffer_LAMP_C2_PTM_04 : ComBuffer;
	SerialTXBuffer_LAMP_C2_PTM_04 : ComBuffer;	
	SerialRXBuffer_LAMP_ROUGH_PTM_01 : ComBuffer;
	SerialTXBuffer_LAMP_ROUGH_PTM_01 : ComBuffer;	
	SerialRXBuffer_LAMP_C1_PTM_01 : ComBuffer;
	SerialTXBuffer_LAMP_C1_PTM_01 : ComBuffer;	
	SerialRXBuffer_LAMP_CATCH_PTM_01 : ComBuffer;
	SerialTXBuffer_LAMP_CATCH_PTM_01 : ComBuffer;	
	SerialRXBuffer_LAMP_CATCH_PTM_02 : ComBuffer;
	SerialTXBuffer_LAMP_CATCH_PTM_02 : ComBuffer;

// Cluster Source LV17 configuration
    SerialTXBuffer_LAMP_CLSTR1_PTM_01 : ComBuffer;	
	SerialRXBuffer_LAMP_CLSTR1_PTM_01 : ComBuffer;
	SerialTXBuffer_LAMP_CLSTR1_PTM_02 : ComBuffer;	
	SerialRXBuffer_LAMP_CLSTR1_PTM_02 : ComBuffer;
	SerialTXBuffer_LAMP_CLSTR1_PTM_03 : ComBuffer;	
	SerialRXBuffer_LAMP_CLSTR1_PTM_03 : ComBuffer;
(*	
	SerialRXBuffer_KTOF_PTM_01 : ComBuffer;
	SerialTXBuffer_KTOF_PTM_01 : ComBuffer;
*)	
	
	// Serial Terminal
	fbSerialLineControl_LAMP_C2_PTM_01: SerialLineControl;
	fbSerialLineControl_LAMP_C2_PTM_02: SerialLineControl;
	fbSerialLineControl_LAMP_C2_PTM_03: SerialLineControl;
	fbSerialLineControl_LAMP_C2_PTM_04: SerialLineControl;
	fbSerialLineControl_LAMP_ROUGH_PTM_01: SerialLineControl;
	fbSerialLineControl_LAMP_C1_PTM_01: SerialLineControl;
	fbSerialLineControl_LAMP_CATCH_PTM_01: SerialLineControl;
	fbSerialLineControl_LAMP_CATCH_PTM_02: SerialLineControl;
	fbSerialLineControl_LAMP_CLSTR1_PTM_01: SerialLineControl;
	fbSerialLineControl_LAMP_CLSTR1_PTM_02: SerialLineControl;
	fbSerialLineControl_LAMP_CLSTR1_PTM_03: SerialLineControl;
//	fbSerialLineControl_KTOF_PTM_01: SerialLineControl;
	
	//SERIAL IO
	{attribute	'TcLinkTo'	:=	'.Status:=TIIB[LAMP_PNL1_EP03_EP6002-0002]^COM TxPDO-Map Inputs Channel 1^Status;
								 .D[0]:=TIIB[LAMP_PNL1_EP03_EP6002-0002]^COM TxPDO-Map Inputs Channel 1^Data In 0;
								 .D[1]:=TIIB[LAMP_PNL1_EP03_EP6002-0002]^COM TxPDO-Map Inputs Channel 1^Data In 1;
								 .D[2]:=TIIB[LAMP_PNL1_EP03_EP6002-0002]^COM TxPDO-Map Inputs Channel 1^Data In 2;
								 .D[3]:=TIIB[LAMP_PNL1_EP03_EP6002-0002]^COM TxPDO-Map Inputs Channel 1^Data In 3;
								 .D[4]:=TIIB[LAMP_PNL1_EP03_EP6002-0002]^COM TxPDO-Map Inputs Channel 1^Data In 4;
								 .D[5]:=TIIB[LAMP_PNL1_EP03_EP6002-0002]^COM TxPDO-Map Inputs Channel 1^Data In 5;
								 .D[6]:=TIIB[LAMP_PNL1_EP03_EP6002-0002]^COM TxPDO-Map Inputs Channel 1^Data In 6;
								 .D[7]:=TIIB[LAMP_PNL1_EP03_EP6002-0002]^COM TxPDO-Map Inputs Channel 1^Data In 7;
								 .D[8]:=TIIB[LAMP_PNL1_EP03_EP6002-0002]^COM TxPDO-Map Inputs Channel 1^Data In 8;
								 .D[9]:=TIIB[LAMP_PNL1_EP03_EP6002-0002]^COM TxPDO-Map Inputs Channel 1^Data In 9;
								 .D[10]:=TIIB[LAMP_PNL1_EP03_EP6002-0002]^COM TxPDO-Map Inputs Channel 1^Data In 10;
								 .D[11]:=TIIB[LAMP_PNL1_EP03_EP6002-0002]^COM TxPDO-Map Inputs Channel 1^Data In 11;
								 .D[12]:=TIIB[LAMP_PNL1_EP03_EP6002-0002]^COM TxPDO-Map Inputs Channel 1^Data In 12;
								 .D[13]:=TIIB[LAMP_PNL1_EP03_EP6002-0002]^COM TxPDO-Map Inputs Channel 1^Data In 13;
								 .D[14]:=TIIB[LAMP_PNL1_EP03_EP6002-0002]^COM TxPDO-Map Inputs Channel 1^Data In 14;
								 .D[15]:=TIIB[LAMP_PNL1_EP03_EP6002-0002]^COM TxPDO-Map Inputs Channel 1^Data In 15;
								 .D[16]:=TIIB[LAMP_PNL1_EP03_EP6002-0002]^COM TxPDO-Map Inputs Channel 1^Data In 16;
								 .D[17]:=TIIB[LAMP_PNL1_EP03_EP6002-0002]^COM TxPDO-Map Inputs Channel 1^Data In 17;
								 .D[18]:=TIIB[LAMP_PNL1_EP03_EP6002-0002]^COM TxPDO-Map Inputs Channel 1^Data In 18;
								 .D[19]:=TIIB[LAMP_PNL1_EP03_EP6002-0002]^COM TxPDO-Map Inputs Channel 1^Data In 19;
								 .D[20]:=TIIB[LAMP_PNL1_EP03_EP6002-0002]^COM TxPDO-Map Inputs Channel 1^Data In 20;
								 .D[21]:=TIIB[LAMP_PNL1_EP03_EP6002-0002]^COM TxPDO-Map Inputs Channel 1^Data In 21
	'}
	stComIn_LAMP_C2_PTM_01		AT %I*	:	EL6inData22B;
	
	{attribute	'TcLinkTo'	:=	'.Ctrl:=TIIB[LAMP_PNL1_EP03_EP6002-0002]^COM RxPDO-Map Outputs Channel 1^Ctrl;
								 .D[0]:=TIIB[LAMP_PNL1_EP03_EP6002-0002]^COM RxPDO-Map Outputs Channel 1^Data Out 0;
								 .D[1]:=TIIB[LAMP_PNL1_EP03_EP6002-0002]^COM RxPDO-Map Outputs Channel 1^Data Out 1;
								 .D[2]:=TIIB[LAMP_PNL1_EP03_EP6002-0002]^COM RxPDO-Map Outputs Channel 1^Data Out 2;
								 .D[3]:=TIIB[LAMP_PNL1_EP03_EP6002-0002]^COM RxPDO-Map Outputs Channel 1^Data Out 3;
								 .D[4]:=TIIB[LAMP_PNL1_EP03_EP6002-0002]^COM RxPDO-Map Outputs Channel 1^Data Out 4;
								 .D[5]:=TIIB[LAMP_PNL1_EP03_EP6002-0002]^COM RxPDO-Map Outputs Channel 1^Data Out 5;
								 .D[6]:=TIIB[LAMP_PNL1_EP03_EP6002-0002]^COM RxPDO-Map Outputs Channel 1^Data Out 6;
								 .D[7]:=TIIB[LAMP_PNL1_EP03_EP6002-0002]^COM RxPDO-Map Outputs Channel 1^Data Out 7;
								 .D[8]:=TIIB[LAMP_PNL1_EP03_EP6002-0002]^COM RxPDO-Map Outputs Channel 1^Data Out 8;
								 .D[9]:=TIIB[LAMP_PNL1_EP03_EP6002-0002]^COM RxPDO-Map Outputs Channel 1^Data Out 9;
								 .D[10]:=TIIB[LAMP_PNL1_EP03_EP6002-0002]^COM RxPDO-Map Outputs Channel 1^Data Out 10;
								 .D[11]:=TIIB[LAMP_PNL1_EP03_EP6002-0002]^COM RxPDO-Map Outputs Channel 1^Data Out 11;
								 .D[12]:=TIIB[LAMP_PNL1_EP03_EP6002-0002]^COM RxPDO-Map Outputs Channel 1^Data Out 12;
								 .D[13]:=TIIB[LAMP_PNL1_EP03_EP6002-0002]^COM RxPDO-Map Outputs Channel 1^Data Out 13;
								 .D[14]:=TIIB[LAMP_PNL1_EP03_EP6002-0002]^COM RxPDO-Map Outputs Channel 1^Data Out 14;
								 .D[15]:=TIIB[LAMP_PNL1_EP03_EP6002-0002]^COM RxPDO-Map Outputs Channel 1^Data Out 15;
								 .D[16]:=TIIB[LAMP_PNL1_EP03_EP6002-0002]^COM RxPDO-Map Outputs Channel 1^Data Out 16;
								 .D[17]:=TIIB[LAMP_PNL1_EP03_EP6002-0002]^COM RxPDO-Map Outputs Channel 1^Data Out 17;
								 .D[18]:=TIIB[LAMP_PNL1_EP03_EP6002-0002]^COM RxPDO-Map Outputs Channel 1^Data Out 18;
								 .D[19]:=TIIB[LAMP_PNL1_EP03_EP6002-0002]^COM RxPDO-Map Outputs Channel 1^Data Out 19;
								 .D[20]:=TIIB[LAMP_PNL1_EP03_EP6002-0002]^COM RxPDO-Map Outputs Channel 1^Data Out 20;
								 .D[21]:=TIIB[LAMP_PNL1_EP03_EP6002-0002]^COM RxPDO-Map Outputs Channel 1^Data Out 21
	'}
	stComOut_LAMP_C2_PTM_01		AT %Q*	:	EL6outData22B;
	
	{attribute	'TcLinkTo'	:=	'.Status:=TIIB[LAMP_PNL1_EP03_EP6002-0002]^COM TxPDO-Map Inputs Channel 2^Status;
								 .D[0]:=TIIB[LAMP_PNL1_EP03_EP6002-0002]^COM TxPDO-Map Inputs Channel 2^Data In 0;
								 .D[1]:=TIIB[LAMP_PNL1_EP03_EP6002-0002]^COM TxPDO-Map Inputs Channel 2^Data In 1;
								 .D[2]:=TIIB[LAMP_PNL1_EP03_EP6002-0002]^COM TxPDO-Map Inputs Channel 2^Data In 2;
								 .D[3]:=TIIB[LAMP_PNL1_EP03_EP6002-0002]^COM TxPDO-Map Inputs Channel 2^Data In 3;
								 .D[4]:=TIIB[LAMP_PNL1_EP03_EP6002-0002]^COM TxPDO-Map Inputs Channel 2^Data In 4;
								 .D[5]:=TIIB[LAMP_PNL1_EP03_EP6002-0002]^COM TxPDO-Map Inputs Channel 2^Data In 5;
								 .D[6]:=TIIB[LAMP_PNL1_EP03_EP6002-0002]^COM TxPDO-Map Inputs Channel 2^Data In 6;
								 .D[7]:=TIIB[LAMP_PNL1_EP03_EP6002-0002]^COM TxPDO-Map Inputs Channel 2^Data In 7;
								 .D[8]:=TIIB[LAMP_PNL1_EP03_EP6002-0002]^COM TxPDO-Map Inputs Channel 2^Data In 8;
								 .D[9]:=TIIB[LAMP_PNL1_EP03_EP6002-0002]^COM TxPDO-Map Inputs Channel 2^Data In 9;
								 .D[10]:=TIIB[LAMP_PNL1_EP03_EP6002-0002]^COM TxPDO-Map Inputs Channel 2^Data In 10;
								 .D[11]:=TIIB[LAMP_PNL1_EP03_EP6002-0002]^COM TxPDO-Map Inputs Channel 2^Data In 11;
								 .D[12]:=TIIB[LAMP_PNL1_EP03_EP6002-0002]^COM TxPDO-Map Inputs Channel 2^Data In 12;
								 .D[13]:=TIIB[LAMP_PNL1_EP03_EP6002-0002]^COM TxPDO-Map Inputs Channel 2^Data In 13;
								 .D[14]:=TIIB[LAMP_PNL1_EP03_EP6002-0002]^COM TxPDO-Map Inputs Channel 2^Data In 14;
								 .D[15]:=TIIB[LAMP_PNL1_EP03_EP6002-0002]^COM TxPDO-Map Inputs Channel 2^Data In 15;
								 .D[16]:=TIIB[LAMP_PNL1_EP03_EP6002-0002]^COM TxPDO-Map Inputs Channel 2^Data In 16;
								 .D[17]:=TIIB[LAMP_PNL1_EP03_EP6002-0002]^COM TxPDO-Map Inputs Channel 2^Data In 17;
								 .D[18]:=TIIB[LAMP_PNL1_EP03_EP6002-0002]^COM TxPDO-Map Inputs Channel 2^Data In 18;
								 .D[19]:=TIIB[LAMP_PNL1_EP03_EP6002-0002]^COM TxPDO-Map Inputs Channel 2^Data In 19;
								 .D[20]:=TIIB[LAMP_PNL1_EP03_EP6002-0002]^COM TxPDO-Map Inputs Channel 2^Data In 20;
								 .D[21]:=TIIB[LAMP_PNL1_EP03_EP6002-0002]^COM TxPDO-Map Inputs Channel 2^Data In 21
	'}
	stComIn_LAMP_C2_PTM_02		AT %I*	:	EL6inData22B;
	
	{attribute	'TcLinkTo'	:=	'.Ctrl:=TIIB[LAMP_PNL1_EP03_EP6002-0002]^COM RxPDO-Map Outputs Channel 2^Ctrl;
								 .D[0]:=TIIB[LAMP_PNL1_EP03_EP6002-0002]^COM RxPDO-Map Outputs Channel 2^Data Out 0;
								 .D[1]:=TIIB[LAMP_PNL1_EP03_EP6002-0002]^COM RxPDO-Map Outputs Channel 2^Data Out 1;
								 .D[2]:=TIIB[LAMP_PNL1_EP03_EP6002-0002]^COM RxPDO-Map Outputs Channel 2^Data Out 2;
								 .D[3]:=TIIB[LAMP_PNL1_EP03_EP6002-0002]^COM RxPDO-Map Outputs Channel 2^Data Out 3;
								 .D[4]:=TIIB[LAMP_PNL1_EP03_EP6002-0002]^COM RxPDO-Map Outputs Channel 2^Data Out 4;
								 .D[5]:=TIIB[LAMP_PNL1_EP03_EP6002-0002]^COM RxPDO-Map Outputs Channel 2^Data Out 5;
								 .D[6]:=TIIB[LAMP_PNL1_EP03_EP6002-0002]^COM RxPDO-Map Outputs Channel 2^Data Out 6;
								 .D[7]:=TIIB[LAMP_PNL1_EP03_EP6002-0002]^COM RxPDO-Map Outputs Channel 2^Data Out 7;
								 .D[8]:=TIIB[LAMP_PNL1_EP03_EP6002-0002]^COM RxPDO-Map Outputs Channel 2^Data Out 8;
								 .D[9]:=TIIB[LAMP_PNL1_EP03_EP6002-0002]^COM RxPDO-Map Outputs Channel 2^Data Out 9;
								 .D[10]:=TIIB[LAMP_PNL1_EP03_EP6002-0002]^COM RxPDO-Map Outputs Channel 2^Data Out 10;
								 .D[11]:=TIIB[LAMP_PNL1_EP03_EP6002-0002]^COM RxPDO-Map Outputs Channel 2^Data Out 11;
								 .D[12]:=TIIB[LAMP_PNL1_EP03_EP6002-0002]^COM RxPDO-Map Outputs Channel 2^Data Out 12;
								 .D[13]:=TIIB[LAMP_PNL1_EP03_EP6002-0002]^COM RxPDO-Map Outputs Channel 2^Data Out 13;
								 .D[14]:=TIIB[LAMP_PNL1_EP03_EP6002-0002]^COM RxPDO-Map Outputs Channel 2^Data Out 14;
								 .D[15]:=TIIB[LAMP_PNL1_EP03_EP6002-0002]^COM RxPDO-Map Outputs Channel 2^Data Out 15;
								 .D[16]:=TIIB[LAMP_PNL1_EP03_EP6002-0002]^COM RxPDO-Map Outputs Channel 2^Data Out 16;
								 .D[17]:=TIIB[LAMP_PNL1_EP03_EP6002-0002]^COM RxPDO-Map Outputs Channel 2^Data Out 17;
								 .D[18]:=TIIB[LAMP_PNL1_EP03_EP6002-0002]^COM RxPDO-Map Outputs Channel 2^Data Out 18;
								 .D[19]:=TIIB[LAMP_PNL1_EP03_EP6002-0002]^COM RxPDO-Map Outputs Channel 2^Data Out 19;
								 .D[20]:=TIIB[LAMP_PNL1_EP03_EP6002-0002]^COM RxPDO-Map Outputs Channel 2^Data Out 20;
								 .D[21]:=TIIB[LAMP_PNL1_EP03_EP6002-0002]^COM RxPDO-Map Outputs Channel 2^Data Out 21
	'}
	stComOut_LAMP_C2_PTM_02		AT %Q*	:	EL6outData22B;
	
	{attribute	'TcLinkTo'	:=	'.Status:=TIIB[LAMP_PNL1_EP06_EP6002-0002]^COM TxPDO-Map Inputs Channel 1^Status;
								 .D[0]:=TIIB[LAMP_PNL1_EP06_EP6002-0002]^COM TxPDO-Map Inputs Channel 1^Data In 0;
								 .D[1]:=TIIB[LAMP_PNL1_EP06_EP6002-0002]^COM TxPDO-Map Inputs Channel 1^Data In 1;
								 .D[2]:=TIIB[LAMP_PNL1_EP06_EP6002-0002]^COM TxPDO-Map Inputs Channel 1^Data In 2;
								 .D[3]:=TIIB[LAMP_PNL1_EP06_EP6002-0002]^COM TxPDO-Map Inputs Channel 1^Data In 3;
								 .D[4]:=TIIB[LAMP_PNL1_EP06_EP6002-0002]^COM TxPDO-Map Inputs Channel 1^Data In 4;
								 .D[5]:=TIIB[LAMP_PNL1_EP06_EP6002-0002]^COM TxPDO-Map Inputs Channel 1^Data In 5;
								 .D[6]:=TIIB[LAMP_PNL1_EP06_EP6002-0002]^COM TxPDO-Map Inputs Channel 1^Data In 6;
								 .D[7]:=TIIB[LAMP_PNL1_EP06_EP6002-0002]^COM TxPDO-Map Inputs Channel 1^Data In 7;
								 .D[8]:=TIIB[LAMP_PNL1_EP06_EP6002-0002]^COM TxPDO-Map Inputs Channel 1^Data In 8;
								 .D[9]:=TIIB[LAMP_PNL1_EP06_EP6002-0002]^COM TxPDO-Map Inputs Channel 1^Data In 9;
								 .D[10]:=TIIB[LAMP_PNL1_EP06_EP6002-0002]^COM TxPDO-Map Inputs Channel 1^Data In 10;
								 .D[11]:=TIIB[LAMP_PNL1_EP06_EP6002-0002]^COM TxPDO-Map Inputs Channel 1^Data In 11;
								 .D[12]:=TIIB[LAMP_PNL1_EP06_EP6002-0002]^COM TxPDO-Map Inputs Channel 1^Data In 12;
								 .D[13]:=TIIB[LAMP_PNL1_EP06_EP6002-0002]^COM TxPDO-Map Inputs Channel 1^Data In 13;
								 .D[14]:=TIIB[LAMP_PNL1_EP06_EP6002-0002]^COM TxPDO-Map Inputs Channel 1^Data In 14;
								 .D[15]:=TIIB[LAMP_PNL1_EP06_EP6002-0002]^COM TxPDO-Map Inputs Channel 1^Data In 15;
								 .D[16]:=TIIB[LAMP_PNL1_EP06_EP6002-0002]^COM TxPDO-Map Inputs Channel 1^Data In 16;
								 .D[17]:=TIIB[LAMP_PNL1_EP06_EP6002-0002]^COM TxPDO-Map Inputs Channel 1^Data In 17;
								 .D[18]:=TIIB[LAMP_PNL1_EP06_EP6002-0002]^COM TxPDO-Map Inputs Channel 1^Data In 18;
								 .D[19]:=TIIB[LAMP_PNL1_EP06_EP6002-0002]^COM TxPDO-Map Inputs Channel 1^Data In 19;
								 .D[20]:=TIIB[LAMP_PNL1_EP06_EP6002-0002]^COM TxPDO-Map Inputs Channel 1^Data In 20;
								 .D[21]:=TIIB[LAMP_PNL1_EP06_EP6002-0002]^COM TxPDO-Map Inputs Channel 1^Data In 21
	'}
	stComIn_LAMP_C2_PTM_03		AT %I*	:	EL6inData22B;
	
	{attribute	'TcLinkTo'	:=	'.Ctrl:=TIIB[LAMP_PNL1_EP06_EP6002-0002]^COM RxPDO-Map Outputs Channel 1^Ctrl;
								 .D[0]:=TIIB[LAMP_PNL1_EP06_EP6002-0002]^COM RxPDO-Map Outputs Channel 1^Data Out 0;
								 .D[1]:=TIIB[LAMP_PNL1_EP06_EP6002-0002]^COM RxPDO-Map Outputs Channel 1^Data Out 1;
								 .D[2]:=TIIB[LAMP_PNL1_EP06_EP6002-0002]^COM RxPDO-Map Outputs Channel 1^Data Out 2;
								 .D[3]:=TIIB[LAMP_PNL1_EP06_EP6002-0002]^COM RxPDO-Map Outputs Channel 1^Data Out 3;
								 .D[4]:=TIIB[LAMP_PNL1_EP06_EP6002-0002]^COM RxPDO-Map Outputs Channel 1^Data Out 4;
								 .D[5]:=TIIB[LAMP_PNL1_EP06_EP6002-0002]^COM RxPDO-Map Outputs Channel 1^Data Out 5;
								 .D[6]:=TIIB[LAMP_PNL1_EP06_EP6002-0002]^COM RxPDO-Map Outputs Channel 1^Data Out 6;
								 .D[7]:=TIIB[LAMP_PNL1_EP06_EP6002-0002]^COM RxPDO-Map Outputs Channel 1^Data Out 7;
								 .D[8]:=TIIB[LAMP_PNL1_EP06_EP6002-0002]^COM RxPDO-Map Outputs Channel 1^Data Out 8;
								 .D[9]:=TIIB[LAMP_PNL1_EP06_EP6002-0002]^COM RxPDO-Map Outputs Channel 1^Data Out 9;
								 .D[10]:=TIIB[LAMP_PNL1_EP06_EP6002-0002]^COM RxPDO-Map Outputs Channel 1^Data Out 10;
								 .D[11]:=TIIB[LAMP_PNL1_EP06_EP6002-0002]^COM RxPDO-Map Outputs Channel 1^Data Out 11;
								 .D[12]:=TIIB[LAMP_PNL1_EP06_EP6002-0002]^COM RxPDO-Map Outputs Channel 1^Data Out 12;
								 .D[13]:=TIIB[LAMP_PNL1_EP06_EP6002-0002]^COM RxPDO-Map Outputs Channel 1^Data Out 13;
								 .D[14]:=TIIB[LAMP_PNL1_EP06_EP6002-0002]^COM RxPDO-Map Outputs Channel 1^Data Out 14;
								 .D[15]:=TIIB[LAMP_PNL1_EP06_EP6002-0002]^COM RxPDO-Map Outputs Channel 1^Data Out 15;
								 .D[16]:=TIIB[LAMP_PNL1_EP06_EP6002-0002]^COM RxPDO-Map Outputs Channel 1^Data Out 16;
								 .D[17]:=TIIB[LAMP_PNL1_EP06_EP6002-0002]^COM RxPDO-Map Outputs Channel 1^Data Out 17;
								 .D[18]:=TIIB[LAMP_PNL1_EP06_EP6002-0002]^COM RxPDO-Map Outputs Channel 1^Data Out 18;
								 .D[19]:=TIIB[LAMP_PNL1_EP06_EP6002-0002]^COM RxPDO-Map Outputs Channel 1^Data Out 19;
								 .D[20]:=TIIB[LAMP_PNL1_EP06_EP6002-0002]^COM RxPDO-Map Outputs Channel 1^Data Out 20;
								 .D[21]:=TIIB[LAMP_PNL1_EP06_EP6002-0002]^COM RxPDO-Map Outputs Channel 1^Data Out 21
	'}
	stComOut_LAMP_C2_PTM_03		AT %Q*	:	EL6outData22B;
	
	{attribute	'TcLinkTo'	:=	'.Status:=TIIB[LAMP_PNL1_EP06_EP6002-0002]^COM TxPDO-Map Inputs Channel 2^Status;
								 .D[0]:=TIIB[LAMP_PNL1_EP06_EP6002-0002]^COM TxPDO-Map Inputs Channel 2^Data In 0;
								 .D[1]:=TIIB[LAMP_PNL1_EP06_EP6002-0002]^COM TxPDO-Map Inputs Channel 2^Data In 1;
								 .D[2]:=TIIB[LAMP_PNL1_EP06_EP6002-0002]^COM TxPDO-Map Inputs Channel 2^Data In 2;
								 .D[3]:=TIIB[LAMP_PNL1_EP06_EP6002-0002]^COM TxPDO-Map Inputs Channel 2^Data In 3;
								 .D[4]:=TIIB[LAMP_PNL1_EP06_EP6002-0002]^COM TxPDO-Map Inputs Channel 2^Data In 4;
								 .D[5]:=TIIB[LAMP_PNL1_EP06_EP6002-0002]^COM TxPDO-Map Inputs Channel 2^Data In 5;
								 .D[6]:=TIIB[LAMP_PNL1_EP06_EP6002-0002]^COM TxPDO-Map Inputs Channel 2^Data In 6;
								 .D[7]:=TIIB[LAMP_PNL1_EP06_EP6002-0002]^COM TxPDO-Map Inputs Channel 2^Data In 7;
								 .D[8]:=TIIB[LAMP_PNL1_EP06_EP6002-0002]^COM TxPDO-Map Inputs Channel 2^Data In 8;
								 .D[9]:=TIIB[LAMP_PNL1_EP06_EP6002-0002]^COM TxPDO-Map Inputs Channel 2^Data In 9;
								 .D[10]:=TIIB[LAMP_PNL1_EP06_EP6002-0002]^COM TxPDO-Map Inputs Channel 2^Data In 10;
								 .D[11]:=TIIB[LAMP_PNL1_EP06_EP6002-0002]^COM TxPDO-Map Inputs Channel 2^Data In 11;
								 .D[12]:=TIIB[LAMP_PNL1_EP06_EP6002-0002]^COM TxPDO-Map Inputs Channel 2^Data In 12;
								 .D[13]:=TIIB[LAMP_PNL1_EP06_EP6002-0002]^COM TxPDO-Map Inputs Channel 2^Data In 13;
								 .D[14]:=TIIB[LAMP_PNL1_EP06_EP6002-0002]^COM TxPDO-Map Inputs Channel 2^Data In 14;
								 .D[15]:=TIIB[LAMP_PNL1_EP06_EP6002-0002]^COM TxPDO-Map Inputs Channel 2^Data In 15;
								 .D[16]:=TIIB[LAMP_PNL1_EP06_EP6002-0002]^COM TxPDO-Map Inputs Channel 2^Data In 16;
								 .D[17]:=TIIB[LAMP_PNL1_EP06_EP6002-0002]^COM TxPDO-Map Inputs Channel 2^Data In 17;
								 .D[18]:=TIIB[LAMP_PNL1_EP06_EP6002-0002]^COM TxPDO-Map Inputs Channel 2^Data In 18;
								 .D[19]:=TIIB[LAMP_PNL1_EP06_EP6002-0002]^COM TxPDO-Map Inputs Channel 2^Data In 19;
								 .D[20]:=TIIB[LAMP_PNL1_EP06_EP6002-0002]^COM TxPDO-Map Inputs Channel 2^Data In 20;
								 .D[21]:=TIIB[LAMP_PNL1_EP06_EP6002-0002]^COM TxPDO-Map Inputs Channel 2^Data In 21
	'}
	stComIn_LAMP_C2_PTM_04		AT %I*	:	EL6inData22B;
	
	{attribute	'TcLinkTo'	:=	'.Ctrl:=TIIB[LAMP_PNL1_EP06_EP6002-0002]^COM RxPDO-Map Outputs Channel 2^Ctrl;
								 .D[0]:=TIIB[LAMP_PNL1_EP06_EP6002-0002]^COM RxPDO-Map Outputs Channel 2^Data Out 0;
								 .D[1]:=TIIB[LAMP_PNL1_EP06_EP6002-0002]^COM RxPDO-Map Outputs Channel 2^Data Out 1;
								 .D[2]:=TIIB[LAMP_PNL1_EP06_EP6002-0002]^COM RxPDO-Map Outputs Channel 2^Data Out 2;
								 .D[3]:=TIIB[LAMP_PNL1_EP06_EP6002-0002]^COM RxPDO-Map Outputs Channel 2^Data Out 3;
								 .D[4]:=TIIB[LAMP_PNL1_EP06_EP6002-0002]^COM RxPDO-Map Outputs Channel 2^Data Out 4;
								 .D[5]:=TIIB[LAMP_PNL1_EP06_EP6002-0002]^COM RxPDO-Map Outputs Channel 2^Data Out 5;
								 .D[6]:=TIIB[LAMP_PNL1_EP06_EP6002-0002]^COM RxPDO-Map Outputs Channel 2^Data Out 6;
								 .D[7]:=TIIB[LAMP_PNL1_EP06_EP6002-0002]^COM RxPDO-Map Outputs Channel 2^Data Out 7;
								 .D[8]:=TIIB[LAMP_PNL1_EP06_EP6002-0002]^COM RxPDO-Map Outputs Channel 2^Data Out 8;
								 .D[9]:=TIIB[LAMP_PNL1_EP06_EP6002-0002]^COM RxPDO-Map Outputs Channel 2^Data Out 9;
								 .D[10]:=TIIB[LAMP_PNL1_EP06_EP6002-0002]^COM RxPDO-Map Outputs Channel 2^Data Out 10;
								 .D[11]:=TIIB[LAMP_PNL1_EP06_EP6002-0002]^COM RxPDO-Map Outputs Channel 2^Data Out 11;
								 .D[12]:=TIIB[LAMP_PNL1_EP06_EP6002-0002]^COM RxPDO-Map Outputs Channel 2^Data Out 12;
								 .D[13]:=TIIB[LAMP_PNL1_EP06_EP6002-0002]^COM RxPDO-Map Outputs Channel 2^Data Out 13;
								 .D[14]:=TIIB[LAMP_PNL1_EP06_EP6002-0002]^COM RxPDO-Map Outputs Channel 2^Data Out 14;
								 .D[15]:=TIIB[LAMP_PNL1_EP06_EP6002-0002]^COM RxPDO-Map Outputs Channel 2^Data Out 15;
								 .D[16]:=TIIB[LAMP_PNL1_EP06_EP6002-0002]^COM RxPDO-Map Outputs Channel 2^Data Out 16;
								 .D[17]:=TIIB[LAMP_PNL1_EP06_EP6002-0002]^COM RxPDO-Map Outputs Channel 2^Data Out 17;
								 .D[18]:=TIIB[LAMP_PNL1_EP06_EP6002-0002]^COM RxPDO-Map Outputs Channel 2^Data Out 18;
								 .D[19]:=TIIB[LAMP_PNL1_EP06_EP6002-0002]^COM RxPDO-Map Outputs Channel 2^Data Out 19;
								 .D[20]:=TIIB[LAMP_PNL1_EP06_EP6002-0002]^COM RxPDO-Map Outputs Channel 2^Data Out 20;
								 .D[21]:=TIIB[LAMP_PNL1_EP06_EP6002-0002]^COM RxPDO-Map Outputs Channel 2^Data Out 21
	'}
	stComOut_LAMP_C2_PTM_04		AT %Q*	:	EL6outData22B;
	
	{attribute	'TcLinkTo'	:=	'.Status:=TIIB[LAMP_PNL2_EP15_EP6002-0002]^COM TxPDO-Map Inputs Channel 1^Status;
								 .D[0]:=TIIB[LAMP_PNL2_EP15_EP6002-0002]^COM TxPDO-Map Inputs Channel 1^Data In 0;
								 .D[1]:=TIIB[LAMP_PNL2_EP15_EP6002-0002]^COM TxPDO-Map Inputs Channel 1^Data In 1;
								 .D[2]:=TIIB[LAMP_PNL2_EP15_EP6002-0002]^COM TxPDO-Map Inputs Channel 1^Data In 2;
								 .D[3]:=TIIB[LAMP_PNL2_EP15_EP6002-0002]^COM TxPDO-Map Inputs Channel 1^Data In 3;
								 .D[4]:=TIIB[LAMP_PNL2_EP15_EP6002-0002]^COM TxPDO-Map Inputs Channel 1^Data In 4;
								 .D[5]:=TIIB[LAMP_PNL2_EP15_EP6002-0002]^COM TxPDO-Map Inputs Channel 1^Data In 5;
								 .D[6]:=TIIB[LAMP_PNL2_EP15_EP6002-0002]^COM TxPDO-Map Inputs Channel 1^Data In 6;
								 .D[7]:=TIIB[LAMP_PNL2_EP15_EP6002-0002]^COM TxPDO-Map Inputs Channel 1^Data In 7;
								 .D[8]:=TIIB[LAMP_PNL2_EP15_EP6002-0002]^COM TxPDO-Map Inputs Channel 1^Data In 8;
								 .D[9]:=TIIB[LAMP_PNL2_EP15_EP6002-0002]^COM TxPDO-Map Inputs Channel 1^Data In 9;
								 .D[10]:=TIIB[LAMP_PNL2_EP15_EP6002-0002]^COM TxPDO-Map Inputs Channel 1^Data In 10;
								 .D[11]:=TIIB[LAMP_PNL2_EP15_EP6002-0002]^COM TxPDO-Map Inputs Channel 1^Data In 11;
								 .D[12]:=TIIB[LAMP_PNL2_EP15_EP6002-0002]^COM TxPDO-Map Inputs Channel 1^Data In 12;
								 .D[13]:=TIIB[LAMP_PNL2_EP15_EP6002-0002]^COM TxPDO-Map Inputs Channel 1^Data In 13;
								 .D[14]:=TIIB[LAMP_PNL2_EP15_EP6002-0002]^COM TxPDO-Map Inputs Channel 1^Data In 14;
								 .D[15]:=TIIB[LAMP_PNL2_EP15_EP6002-0002]^COM TxPDO-Map Inputs Channel 1^Data In 15;
								 .D[16]:=TIIB[LAMP_PNL2_EP15_EP6002-0002]^COM TxPDO-Map Inputs Channel 1^Data In 16;
								 .D[17]:=TIIB[LAMP_PNL2_EP15_EP6002-0002]^COM TxPDO-Map Inputs Channel 1^Data In 17;
								 .D[18]:=TIIB[LAMP_PNL2_EP15_EP6002-0002]^COM TxPDO-Map Inputs Channel 1^Data In 18;
								 .D[19]:=TIIB[LAMP_PNL2_EP15_EP6002-0002]^COM TxPDO-Map Inputs Channel 1^Data In 19;
								 .D[20]:=TIIB[LAMP_PNL2_EP15_EP6002-0002]^COM TxPDO-Map Inputs Channel 1^Data In 20;
								 .D[21]:=TIIB[LAMP_PNL2_EP15_EP6002-0002]^COM TxPDO-Map Inputs Channel 1^Data In 21
	'}
	stComIn_LAMP_ROUGH_PTM_01		AT %I*	:	EL6inData22B;
	
	{attribute	'TcLinkTo'	:=	'.Ctrl:=TIIB[LAMP_PNL2_EP15_EP6002-0002]^COM RxPDO-Map Outputs Channel 1^Ctrl;
								 .D[0]:=TIIB[LAMP_PNL2_EP15_EP6002-0002]^COM RxPDO-Map Outputs Channel 1^Data Out 0;
								 .D[1]:=TIIB[LAMP_PNL2_EP15_EP6002-0002]^COM RxPDO-Map Outputs Channel 1^Data Out 1;
								 .D[2]:=TIIB[LAMP_PNL2_EP15_EP6002-0002]^COM RxPDO-Map Outputs Channel 1^Data Out 2;
								 .D[3]:=TIIB[LAMP_PNL2_EP15_EP6002-0002]^COM RxPDO-Map Outputs Channel 1^Data Out 3;
								 .D[4]:=TIIB[LAMP_PNL2_EP15_EP6002-0002]^COM RxPDO-Map Outputs Channel 1^Data Out 4;
								 .D[5]:=TIIB[LAMP_PNL2_EP15_EP6002-0002]^COM RxPDO-Map Outputs Channel 1^Data Out 5;
								 .D[6]:=TIIB[LAMP_PNL2_EP15_EP6002-0002]^COM RxPDO-Map Outputs Channel 1^Data Out 6;
								 .D[7]:=TIIB[LAMP_PNL2_EP15_EP6002-0002]^COM RxPDO-Map Outputs Channel 1^Data Out 7;
								 .D[8]:=TIIB[LAMP_PNL2_EP15_EP6002-0002]^COM RxPDO-Map Outputs Channel 1^Data Out 8;
								 .D[9]:=TIIB[LAMP_PNL2_EP15_EP6002-0002]^COM RxPDO-Map Outputs Channel 1^Data Out 9;
								 .D[10]:=TIIB[LAMP_PNL2_EP15_EP6002-0002]^COM RxPDO-Map Outputs Channel 1^Data Out 10;
								 .D[11]:=TIIB[LAMP_PNL2_EP15_EP6002-0002]^COM RxPDO-Map Outputs Channel 1^Data Out 11;
								 .D[12]:=TIIB[LAMP_PNL2_EP15_EP6002-0002]^COM RxPDO-Map Outputs Channel 1^Data Out 12;
								 .D[13]:=TIIB[LAMP_PNL2_EP15_EP6002-0002]^COM RxPDO-Map Outputs Channel 1^Data Out 13;
								 .D[14]:=TIIB[LAMP_PNL2_EP15_EP6002-0002]^COM RxPDO-Map Outputs Channel 1^Data Out 14;
								 .D[15]:=TIIB[LAMP_PNL2_EP15_EP6002-0002]^COM RxPDO-Map Outputs Channel 1^Data Out 15;
								 .D[16]:=TIIB[LAMP_PNL2_EP15_EP6002-0002]^COM RxPDO-Map Outputs Channel 1^Data Out 16;
								 .D[17]:=TIIB[LAMP_PNL2_EP15_EP6002-0002]^COM RxPDO-Map Outputs Channel 1^Data Out 17;
								 .D[18]:=TIIB[LAMP_PNL2_EP15_EP6002-0002]^COM RxPDO-Map Outputs Channel 1^Data Out 18;
								 .D[19]:=TIIB[LAMP_PNL2_EP15_EP6002-0002]^COM RxPDO-Map Outputs Channel 1^Data Out 19;
								 .D[20]:=TIIB[LAMP_PNL2_EP15_EP6002-0002]^COM RxPDO-Map Outputs Channel 1^Data Out 20;
								 .D[21]:=TIIB[LAMP_PNL2_EP15_EP6002-0002]^COM RxPDO-Map Outputs Channel 1^Data Out 21
	'}
	stComOut_LAMP_ROUGH_PTM_01		AT %Q*	:	EL6outData22B;
	
	{attribute	'TcLinkTo'	:=	'.Status:=TIIB[LAMP_PNL2_EP15_EP6002-0002]^COM TxPDO-Map Inputs Channel 2^Status;
								 .D[0]:=TIIB[LAMP_PNL2_EP15_EP6002-0002]^COM TxPDO-Map Inputs Channel 2^Data In 0;
								 .D[1]:=TIIB[LAMP_PNL2_EP15_EP6002-0002]^COM TxPDO-Map Inputs Channel 2^Data In 1;
								 .D[2]:=TIIB[LAMP_PNL2_EP15_EP6002-0002]^COM TxPDO-Map Inputs Channel 2^Data In 2;
								 .D[3]:=TIIB[LAMP_PNL2_EP15_EP6002-0002]^COM TxPDO-Map Inputs Channel 2^Data In 3;
								 .D[4]:=TIIB[LAMP_PNL2_EP15_EP6002-0002]^COM TxPDO-Map Inputs Channel 2^Data In 4;
								 .D[5]:=TIIB[LAMP_PNL2_EP15_EP6002-0002]^COM TxPDO-Map Inputs Channel 2^Data In 5;
								 .D[6]:=TIIB[LAMP_PNL2_EP15_EP6002-0002]^COM TxPDO-Map Inputs Channel 2^Data In 6;
								 .D[7]:=TIIB[LAMP_PNL2_EP15_EP6002-0002]^COM TxPDO-Map Inputs Channel 2^Data In 7;
								 .D[8]:=TIIB[LAMP_PNL2_EP15_EP6002-0002]^COM TxPDO-Map Inputs Channel 2^Data In 8;
								 .D[9]:=TIIB[LAMP_PNL2_EP15_EP6002-0002]^COM TxPDO-Map Inputs Channel 2^Data In 9;
								 .D[10]:=TIIB[LAMP_PNL2_EP15_EP6002-0002]^COM TxPDO-Map Inputs Channel 2^Data In 10;
								 .D[11]:=TIIB[LAMP_PNL2_EP15_EP6002-0002]^COM TxPDO-Map Inputs Channel 2^Data In 11;
								 .D[12]:=TIIB[LAMP_PNL2_EP15_EP6002-0002]^COM TxPDO-Map Inputs Channel 2^Data In 12;
								 .D[13]:=TIIB[LAMP_PNL2_EP15_EP6002-0002]^COM TxPDO-Map Inputs Channel 2^Data In 13;
								 .D[14]:=TIIB[LAMP_PNL2_EP15_EP6002-0002]^COM TxPDO-Map Inputs Channel 2^Data In 14;
								 .D[15]:=TIIB[LAMP_PNL2_EP15_EP6002-0002]^COM TxPDO-Map Inputs Channel 2^Data In 15;
								 .D[16]:=TIIB[LAMP_PNL2_EP15_EP6002-0002]^COM TxPDO-Map Inputs Channel 2^Data In 16;
								 .D[17]:=TIIB[LAMP_PNL2_EP15_EP6002-0002]^COM TxPDO-Map Inputs Channel 2^Data In 17;
								 .D[18]:=TIIB[LAMP_PNL2_EP15_EP6002-0002]^COM TxPDO-Map Inputs Channel 2^Data In 18;
								 .D[19]:=TIIB[LAMP_PNL2_EP15_EP6002-0002]^COM TxPDO-Map Inputs Channel 2^Data In 19;
								 .D[20]:=TIIB[LAMP_PNL2_EP15_EP6002-0002]^COM TxPDO-Map Inputs Channel 2^Data In 20;
								 .D[21]:=TIIB[LAMP_PNL2_EP15_EP6002-0002]^COM TxPDO-Map Inputs Channel 2^Data In 21
	'}
	stComIn_LAMP_C1_PTM_01		AT %I*	:	EL6inData22B;
	
	{attribute	'TcLinkTo'	:=	'.Ctrl:=TIIB[LAMP_PNL2_EP15_EP6002-0002]^COM RxPDO-Map Outputs Channel 2^Ctrl;
								 .D[0]:=TIIB[LAMP_PNL2_EP15_EP6002-0002]^COM RxPDO-Map Outputs Channel 2^Data Out 0;
								 .D[1]:=TIIB[LAMP_PNL2_EP15_EP6002-0002]^COM RxPDO-Map Outputs Channel 2^Data Out 1;
								 .D[2]:=TIIB[LAMP_PNL2_EP15_EP6002-0002]^COM RxPDO-Map Outputs Channel 2^Data Out 2;
								 .D[3]:=TIIB[LAMP_PNL2_EP15_EP6002-0002]^COM RxPDO-Map Outputs Channel 2^Data Out 3;
								 .D[4]:=TIIB[LAMP_PNL2_EP15_EP6002-0002]^COM RxPDO-Map Outputs Channel 2^Data Out 4;
								 .D[5]:=TIIB[LAMP_PNL2_EP15_EP6002-0002]^COM RxPDO-Map Outputs Channel 2^Data Out 5;
								 .D[6]:=TIIB[LAMP_PNL2_EP15_EP6002-0002]^COM RxPDO-Map Outputs Channel 2^Data Out 6;
								 .D[7]:=TIIB[LAMP_PNL2_EP15_EP6002-0002]^COM RxPDO-Map Outputs Channel 2^Data Out 7;
								 .D[8]:=TIIB[LAMP_PNL2_EP15_EP6002-0002]^COM RxPDO-Map Outputs Channel 2^Data Out 8;
								 .D[9]:=TIIB[LAMP_PNL2_EP15_EP6002-0002]^COM RxPDO-Map Outputs Channel 2^Data Out 9;
								 .D[10]:=TIIB[LAMP_PNL2_EP15_EP6002-0002]^COM RxPDO-Map Outputs Channel 2^Data Out 10;
								 .D[11]:=TIIB[LAMP_PNL2_EP15_EP6002-0002]^COM RxPDO-Map Outputs Channel 2^Data Out 11;
								 .D[12]:=TIIB[LAMP_PNL2_EP15_EP6002-0002]^COM RxPDO-Map Outputs Channel 2^Data Out 12;
								 .D[13]:=TIIB[LAMP_PNL2_EP15_EP6002-0002]^COM RxPDO-Map Outputs Channel 2^Data Out 13;
								 .D[14]:=TIIB[LAMP_PNL2_EP15_EP6002-0002]^COM RxPDO-Map Outputs Channel 2^Data Out 14;
								 .D[15]:=TIIB[LAMP_PNL2_EP15_EP6002-0002]^COM RxPDO-Map Outputs Channel 2^Data Out 15;
								 .D[16]:=TIIB[LAMP_PNL2_EP15_EP6002-0002]^COM RxPDO-Map Outputs Channel 2^Data Out 16;
								 .D[17]:=TIIB[LAMP_PNL2_EP15_EP6002-0002]^COM RxPDO-Map Outputs Channel 2^Data Out 17;
								 .D[18]:=TIIB[LAMP_PNL2_EP15_EP6002-0002]^COM RxPDO-Map Outputs Channel 2^Data Out 18;
								 .D[19]:=TIIB[LAMP_PNL2_EP15_EP6002-0002]^COM RxPDO-Map Outputs Channel 2^Data Out 19;
								 .D[20]:=TIIB[LAMP_PNL2_EP15_EP6002-0002]^COM RxPDO-Map Outputs Channel 2^Data Out 20;
								 .D[21]:=TIIB[LAMP_PNL2_EP15_EP6002-0002]^COM RxPDO-Map Outputs Channel 2^Data Out 21
	'}
	stComOut_LAMP_C1_PTM_01		AT %Q*	:	EL6outData22B;
	
	{attribute	'TcLinkTo'	:=	'.Status:=TIIB[LAMP_PNL2_EP18_EP6002-0002]^COM TxPDO-Map Inputs Channel 1^Status;
								 .D[0]:=TIIB[LAMP_PNL2_EP18_EP6002-0002]^COM TxPDO-Map Inputs Channel 1^Data In 0;
								 .D[1]:=TIIB[LAMP_PNL2_EP18_EP6002-0002]^COM TxPDO-Map Inputs Channel 1^Data In 1;
								 .D[2]:=TIIB[LAMP_PNL2_EP18_EP6002-0002]^COM TxPDO-Map Inputs Channel 1^Data In 2;
								 .D[3]:=TIIB[LAMP_PNL2_EP18_EP6002-0002]^COM TxPDO-Map Inputs Channel 1^Data In 3;
								 .D[4]:=TIIB[LAMP_PNL2_EP18_EP6002-0002]^COM TxPDO-Map Inputs Channel 1^Data In 4;
								 .D[5]:=TIIB[LAMP_PNL2_EP18_EP6002-0002]^COM TxPDO-Map Inputs Channel 1^Data In 5;
								 .D[6]:=TIIB[LAMP_PNL2_EP18_EP6002-0002]^COM TxPDO-Map Inputs Channel 1^Data In 6;
								 .D[7]:=TIIB[LAMP_PNL2_EP18_EP6002-0002]^COM TxPDO-Map Inputs Channel 1^Data In 7;
								 .D[8]:=TIIB[LAMP_PNL2_EP18_EP6002-0002]^COM TxPDO-Map Inputs Channel 1^Data In 8;
								 .D[9]:=TIIB[LAMP_PNL2_EP18_EP6002-0002]^COM TxPDO-Map Inputs Channel 1^Data In 9;
								 .D[10]:=TIIB[LAMP_PNL2_EP18_EP6002-0002]^COM TxPDO-Map Inputs Channel 1^Data In 10;
								 .D[11]:=TIIB[LAMP_PNL2_EP18_EP6002-0002]^COM TxPDO-Map Inputs Channel 1^Data In 11;
								 .D[12]:=TIIB[LAMP_PNL2_EP18_EP6002-0002]^COM TxPDO-Map Inputs Channel 1^Data In 12;
								 .D[13]:=TIIB[LAMP_PNL2_EP18_EP6002-0002]^COM TxPDO-Map Inputs Channel 1^Data In 13;
								 .D[14]:=TIIB[LAMP_PNL2_EP18_EP6002-0002]^COM TxPDO-Map Inputs Channel 1^Data In 14;
								 .D[15]:=TIIB[LAMP_PNL2_EP18_EP6002-0002]^COM TxPDO-Map Inputs Channel 1^Data In 15;
								 .D[16]:=TIIB[LAMP_PNL2_EP18_EP6002-0002]^COM TxPDO-Map Inputs Channel 1^Data In 16;
								 .D[17]:=TIIB[LAMP_PNL2_EP18_EP6002-0002]^COM TxPDO-Map Inputs Channel 1^Data In 17;
								 .D[18]:=TIIB[LAMP_PNL2_EP18_EP6002-0002]^COM TxPDO-Map Inputs Channel 1^Data In 18;
								 .D[19]:=TIIB[LAMP_PNL2_EP18_EP6002-0002]^COM TxPDO-Map Inputs Channel 1^Data In 19;
								 .D[20]:=TIIB[LAMP_PNL2_EP18_EP6002-0002]^COM TxPDO-Map Inputs Channel 1^Data In 20;
								 .D[21]:=TIIB[LAMP_PNL2_EP18_EP6002-0002]^COM TxPDO-Map Inputs Channel 1^Data In 21
	'}
	stComIn_LAMP_CATCH_PTM_01		AT %I*	:	EL6inData22B;
	
	{attribute	'TcLinkTo'	:=	'.Ctrl:=TIIB[LAMP_PNL2_EP18_EP6002-0002]^COM RxPDO-Map Outputs Channel 1^Ctrl;
								 .D[0]:=TIIB[LAMP_PNL2_EP18_EP6002-0002]^COM RxPDO-Map Outputs Channel 1^Data Out 0;
								 .D[1]:=TIIB[LAMP_PNL2_EP18_EP6002-0002]^COM RxPDO-Map Outputs Channel 1^Data Out 1;
								 .D[2]:=TIIB[LAMP_PNL2_EP18_EP6002-0002]^COM RxPDO-Map Outputs Channel 1^Data Out 2;
								 .D[3]:=TIIB[LAMP_PNL2_EP18_EP6002-0002]^COM RxPDO-Map Outputs Channel 1^Data Out 3;
								 .D[4]:=TIIB[LAMP_PNL2_EP18_EP6002-0002]^COM RxPDO-Map Outputs Channel 1^Data Out 4;
								 .D[5]:=TIIB[LAMP_PNL2_EP18_EP6002-0002]^COM RxPDO-Map Outputs Channel 1^Data Out 5;
								 .D[6]:=TIIB[LAMP_PNL2_EP18_EP6002-0002]^COM RxPDO-Map Outputs Channel 1^Data Out 6;
								 .D[7]:=TIIB[LAMP_PNL2_EP18_EP6002-0002]^COM RxPDO-Map Outputs Channel 1^Data Out 7;
								 .D[8]:=TIIB[LAMP_PNL2_EP18_EP6002-0002]^COM RxPDO-Map Outputs Channel 1^Data Out 8;
								 .D[9]:=TIIB[LAMP_PNL2_EP18_EP6002-0002]^COM RxPDO-Map Outputs Channel 1^Data Out 9;
								 .D[10]:=TIIB[LAMP_PNL2_EP18_EP6002-0002]^COM RxPDO-Map Outputs Channel 1^Data Out 10;
								 .D[11]:=TIIB[LAMP_PNL2_EP18_EP6002-0002]^COM RxPDO-Map Outputs Channel 1^Data Out 11;
								 .D[12]:=TIIB[LAMP_PNL2_EP18_EP6002-0002]^COM RxPDO-Map Outputs Channel 1^Data Out 12;
								 .D[13]:=TIIB[LAMP_PNL2_EP18_EP6002-0002]^COM RxPDO-Map Outputs Channel 1^Data Out 13;
								 .D[14]:=TIIB[LAMP_PNL2_EP18_EP6002-0002]^COM RxPDO-Map Outputs Channel 1^Data Out 14;
								 .D[15]:=TIIB[LAMP_PNL2_EP18_EP6002-0002]^COM RxPDO-Map Outputs Channel 1^Data Out 15;
								 .D[16]:=TIIB[LAMP_PNL2_EP18_EP6002-0002]^COM RxPDO-Map Outputs Channel 1^Data Out 16;
								 .D[17]:=TIIB[LAMP_PNL2_EP18_EP6002-0002]^COM RxPDO-Map Outputs Channel 1^Data Out 17;
								 .D[18]:=TIIB[LAMP_PNL2_EP18_EP6002-0002]^COM RxPDO-Map Outputs Channel 1^Data Out 18;
								 .D[19]:=TIIB[LAMP_PNL2_EP18_EP6002-0002]^COM RxPDO-Map Outputs Channel 1^Data Out 19;
								 .D[20]:=TIIB[LAMP_PNL2_EP18_EP6002-0002]^COM RxPDO-Map Outputs Channel 1^Data Out 20;
								 .D[21]:=TIIB[LAMP_PNL2_EP18_EP6002-0002]^COM RxPDO-Map Outputs Channel 1^Data Out 21
	'}
	stComOut_LAMP_CATCH_PTM_01		AT %Q*	:	EL6outData22B;
	
	{attribute	'TcLinkTo'	:=	'.Status:=TIIB[LAMP_PNL2_EP18_EP6002-0002]^COM TxPDO-Map Inputs Channel 2^Status;
								 .D[0]:=TIIB[LAMP_PNL2_EP18_EP6002-0002]^COM TxPDO-Map Inputs Channel 2^Data In 0;
								 .D[1]:=TIIB[LAMP_PNL2_EP18_EP6002-0002]^COM TxPDO-Map Inputs Channel 2^Data In 1;
								 .D[2]:=TIIB[LAMP_PNL2_EP18_EP6002-0002]^COM TxPDO-Map Inputs Channel 2^Data In 2;
								 .D[3]:=TIIB[LAMP_PNL2_EP18_EP6002-0002]^COM TxPDO-Map Inputs Channel 2^Data In 3;
								 .D[4]:=TIIB[LAMP_PNL2_EP18_EP6002-0002]^COM TxPDO-Map Inputs Channel 2^Data In 4;
								 .D[5]:=TIIB[LAMP_PNL2_EP18_EP6002-0002]^COM TxPDO-Map Inputs Channel 2^Data In 5;
								 .D[6]:=TIIB[LAMP_PNL2_EP18_EP6002-0002]^COM TxPDO-Map Inputs Channel 2^Data In 6;
								 .D[7]:=TIIB[LAMP_PNL2_EP18_EP6002-0002]^COM TxPDO-Map Inputs Channel 2^Data In 7;
								 .D[8]:=TIIB[LAMP_PNL2_EP18_EP6002-0002]^COM TxPDO-Map Inputs Channel 2^Data In 8;
								 .D[9]:=TIIB[LAMP_PNL2_EP18_EP6002-0002]^COM TxPDO-Map Inputs Channel 2^Data In 9;
								 .D[10]:=TIIB[LAMP_PNL2_EP18_EP6002-0002]^COM TxPDO-Map Inputs Channel 2^Data In 10;
								 .D[11]:=TIIB[LAMP_PNL2_EP18_EP6002-0002]^COM TxPDO-Map Inputs Channel 2^Data In 11;
								 .D[12]:=TIIB[LAMP_PNL2_EP18_EP6002-0002]^COM TxPDO-Map Inputs Channel 2^Data In 12;
								 .D[13]:=TIIB[LAMP_PNL2_EP18_EP6002-0002]^COM TxPDO-Map Inputs Channel 2^Data In 13;
								 .D[14]:=TIIB[LAMP_PNL2_EP18_EP6002-0002]^COM TxPDO-Map Inputs Channel 2^Data In 14;
								 .D[15]:=TIIB[LAMP_PNL2_EP18_EP6002-0002]^COM TxPDO-Map Inputs Channel 2^Data In 15;
								 .D[16]:=TIIB[LAMP_PNL2_EP18_EP6002-0002]^COM TxPDO-Map Inputs Channel 2^Data In 16;
								 .D[17]:=TIIB[LAMP_PNL2_EP18_EP6002-0002]^COM TxPDO-Map Inputs Channel 2^Data In 17;
								 .D[18]:=TIIB[LAMP_PNL2_EP18_EP6002-0002]^COM TxPDO-Map Inputs Channel 2^Data In 18;
								 .D[19]:=TIIB[LAMP_PNL2_EP18_EP6002-0002]^COM TxPDO-Map Inputs Channel 2^Data In 19;
								 .D[20]:=TIIB[LAMP_PNL2_EP18_EP6002-0002]^COM TxPDO-Map Inputs Channel 2^Data In 20;
								 .D[21]:=TIIB[LAMP_PNL2_EP18_EP6002-0002]^COM TxPDO-Map Inputs Channel 2^Data In 21
	'}
	stComIn_LAMP_CATCH_PTM_02		AT %I*	:	EL6inData22B;
	
	{attribute	'TcLinkTo'	:=	'.Ctrl:=TIIB[LAMP_PNL2_EP18_EP6002-0002]^COM RxPDO-Map Outputs Channel 2^Ctrl;
								 .D[0]:=TIIB[LAMP_PNL2_EP18_EP6002-0002]^COM RxPDO-Map Outputs Channel 2^Data Out 0;
								 .D[1]:=TIIB[LAMP_PNL2_EP18_EP6002-0002]^COM RxPDO-Map Outputs Channel 2^Data Out 1;
								 .D[2]:=TIIB[LAMP_PNL2_EP18_EP6002-0002]^COM RxPDO-Map Outputs Channel 2^Data Out 2;
								 .D[3]:=TIIB[LAMP_PNL2_EP18_EP6002-0002]^COM RxPDO-Map Outputs Channel 2^Data Out 3;
								 .D[4]:=TIIB[LAMP_PNL2_EP18_EP6002-0002]^COM RxPDO-Map Outputs Channel 2^Data Out 4;
								 .D[5]:=TIIB[LAMP_PNL2_EP18_EP6002-0002]^COM RxPDO-Map Outputs Channel 2^Data Out 5;
								 .D[6]:=TIIB[LAMP_PNL2_EP18_EP6002-0002]^COM RxPDO-Map Outputs Channel 2^Data Out 6;
								 .D[7]:=TIIB[LAMP_PNL2_EP18_EP6002-0002]^COM RxPDO-Map Outputs Channel 2^Data Out 7;
								 .D[8]:=TIIB[LAMP_PNL2_EP18_EP6002-0002]^COM RxPDO-Map Outputs Channel 2^Data Out 8;
								 .D[9]:=TIIB[LAMP_PNL2_EP18_EP6002-0002]^COM RxPDO-Map Outputs Channel 2^Data Out 9;
								 .D[10]:=TIIB[LAMP_PNL2_EP18_EP6002-0002]^COM RxPDO-Map Outputs Channel 2^Data Out 10;
								 .D[11]:=TIIB[LAMP_PNL2_EP18_EP6002-0002]^COM RxPDO-Map Outputs Channel 2^Data Out 11;
								 .D[12]:=TIIB[LAMP_PNL2_EP18_EP6002-0002]^COM RxPDO-Map Outputs Channel 2^Data Out 12;
								 .D[13]:=TIIB[LAMP_PNL2_EP18_EP6002-0002]^COM RxPDO-Map Outputs Channel 2^Data Out 13;
								 .D[14]:=TIIB[LAMP_PNL2_EP18_EP6002-0002]^COM RxPDO-Map Outputs Channel 2^Data Out 14;
								 .D[15]:=TIIB[LAMP_PNL2_EP18_EP6002-0002]^COM RxPDO-Map Outputs Channel 2^Data Out 15;
								 .D[16]:=TIIB[LAMP_PNL2_EP18_EP6002-0002]^COM RxPDO-Map Outputs Channel 2^Data Out 16;
								 .D[17]:=TIIB[LAMP_PNL2_EP18_EP6002-0002]^COM RxPDO-Map Outputs Channel 2^Data Out 17;
								 .D[18]:=TIIB[LAMP_PNL2_EP18_EP6002-0002]^COM RxPDO-Map Outputs Channel 2^Data Out 18;
								 .D[19]:=TIIB[LAMP_PNL2_EP18_EP6002-0002]^COM RxPDO-Map Outputs Channel 2^Data Out 19;
								 .D[20]:=TIIB[LAMP_PNL2_EP18_EP6002-0002]^COM RxPDO-Map Outputs Channel 2^Data Out 20;
								 .D[21]:=TIIB[LAMP_PNL2_EP18_EP6002-0002]^COM RxPDO-Map Outputs Channel 2^Data Out 21
	'}
	stComOut_LAMP_CATCH_PTM_02		AT %Q*	:	EL6outData22B;
	
